(* Logix 5000 project; controller cal1615 1756-L62 rev 20.11; software revision 20.05; part 4 of 81 *)

ADD_ON_INSTRUCTION sys_PIDE   (* revision 1.0, vendor Rockwell Automation *)
VAR_IN_OUT
   Autotune_Tag : PIDE_AUTOTUNE; {required}
END_VAR
VAR_INPUT
   ControlAction : BOOL; {required}
END_VAR
VAR_OUTPUT
   CV : REAL; {access Read Only, required}
END_VAR
VAR_INPUT
   CVMax : REAL; {required}
   CVMin : REAL; {required}
END_VAR
VAR_OUTPUT
   Error : REAL; {access Read Only, required}
END_VAR
VAR_INPUT
   Manual_CV : REAL; {required}
   Manual_Mode : BOOL; {required}
END_VAR
VAR_IN_OUT
   PIDE_Tag : PID_ENHANCED; {required}
END_VAR
VAR_INPUT
   PV : REAL; {required}
   PVMax : REAL; {required}
   PVMin : REAL; {required}
   SP : REAL; {required}
END_VAR
VAR
   BAND_01 : FBD_BOOLEAN_AND := (In1 := 1, In2 := 1, In3 := 1, In4 := 1, In5 := 1, In6 := 1, In7 := 1, In8 := 1);
   BNOT_01 : FBD_BOOLEAN_NOT := (In := 1);
   BOR_01 : FBD_BOOLEAN_OR;
   PIDE_Tag_local : PID_ENHANCED := (PVEUMax := 100.0, SPHLimit := 100.0, RatioProg := 1.0, RatioOper := 1.0, RatioHLimit := 1.0, RatioLLimit := 1.0, CVEUMax := 100.0, CVHLimit := 100.0, PVEDerivative := 1, RTSTime := 1);
   TONR_01 : FBD_TIMER;
   PIDE_Tag_01 : PID_ENHANCED := (PVEUMax := 100.0, SPHLimit := 100.0, RatioProg := 1.0, RatioOper := 1.0, RatioHLimit := 1.0, RatioLLimit := 1.0, CVEUMax := 100.0, CVHLimit := 100.0, PVEDerivative := 1, RTSTime := 1);
   BOR_02 : FBD_BOOLEAN_OR;
   TONR_02 : FBD_TIMER;
   BNOT_02 : FBD_BOOLEAN_NOT := (In := 1);
   BAND_02 : FBD_BOOLEAN_AND := (In1 := 1, In2 := 1, In3 := 1, In4 := 1, In5 := 1, In6 := 1, In7 := 1, In8 := 1);
   __l01DD22F71981FEA5 : REAL;
   __l01DD6E4F1981CCC4 : REAL;
   __l01DD12571981E08E : BOOL;
   __l01DD3F0D1981A0DE : REAL;
   __l01DD266519818F93 : BOOL;
   __l01DD4A391981B409 : REAL;
   __l01DD3B8019819839 : REAL;
   __l01DD359A1981A1AC : REAL;
   __l01DD70B31981916B : REAL;
END_VAR

ROUTINE Logic   (* function block diagram *)
   SHEET 1
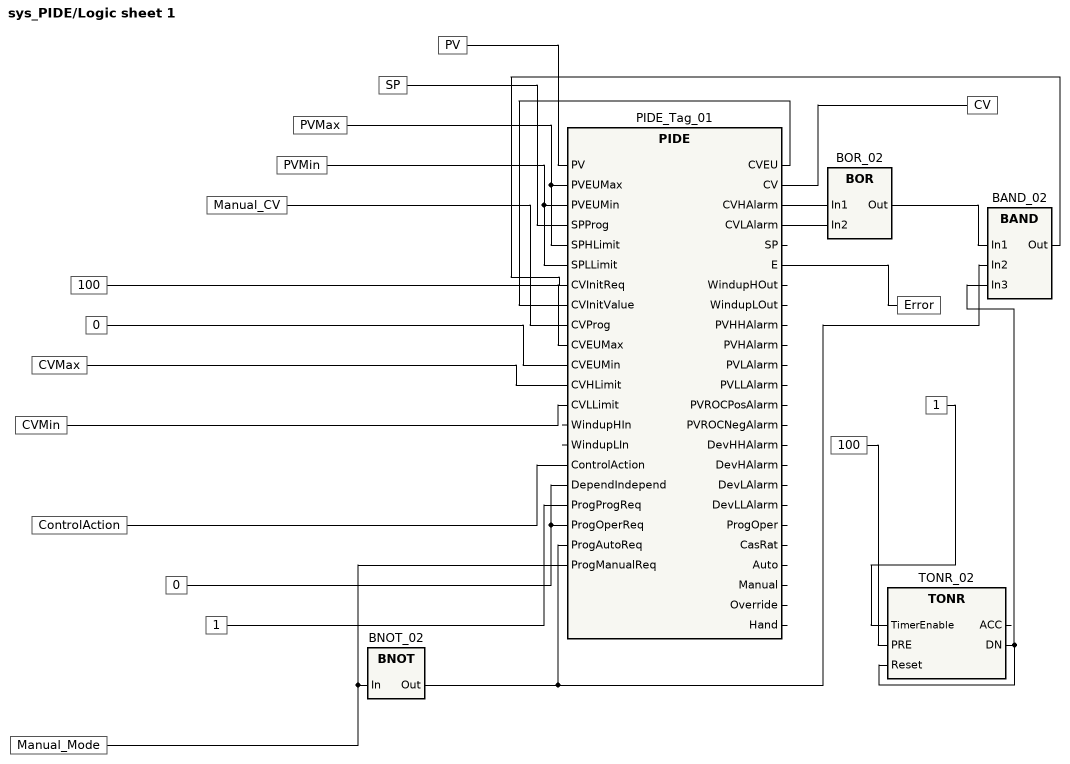
   BNOT_02 : BNOT(In := Manual_Mode);
   PIDE_Tag_01 : PIDE(PV := PV, PVEUMax := PVMax, PVEUMin := PVMin, SPProg := SP, SPHLimit := PVMax, SPLLimit := PVMin, CVInitReq := BAND_02.Out {feedback}, CVInitValue := PIDE_Tag_01.CVEU, CVProg := Manual_CV, CVEUMax := 100, CVEUMin := 0, CVHLimit := CVMax, CVLLimit := CVMin, ControlAction := ControlAction, DependIndepend := 0, ProgProgReq := 1, ProgOperReq := 0, ProgAutoReq := BNOT_02.Out, ProgManualReq := Manual_Mode);   // unwired pins: WindupHIn WindupLIn SP WindupHOut WindupLOut PVHHAlarm PVHAlarm PVLAlarm PVLLAlarm PVROCPosAlarm PVROCNegAlarm DevHHAlarm DevHAlarm DevLAlarm DevLLAlarm ProgOper CasRat Auto Manual Override Hand
   BOR_02 : BOR(In1 := PIDE_Tag_01.CVHAlarm, In2 := PIDE_Tag_01.CVLAlarm);
   Error := PIDE_Tag_01.E;
   CV := PIDE_Tag_01.CV;
   BAND_02 : BAND(In1 := BOR_02.Out, In2 := BNOT_02.Out, In3 := TONR_02.DN {feedback});
   TONR_02 : TONR(TimerEnable := 1, PRE := 100, Reset := TONR_02.DN);   // unwired pins: ACC
END_ROUTINE
END_ADD_ON_INSTRUCTION

ADD_ON_INSTRUCTION sys_Ramp   (* revision 1.0, vendor Rockwell Automation *)
// System Block
// Ramp
VAR_INPUT
   IN_accel_rate : REAL; {required}   // Input Parameter Accel Ramp x/second
   IN_decel_rate : REAL; {required}   // Input Parameter Decel Ramp x/second
   IN_last_scan_s : REAL; {required}   // Input Parameter Last Scan seconds
END_VAR
VAR_IN_OUT
   IN_OUT_ramped_setpoint : REAL; {required}   // Input Output Parameter Ramped Setpoint
END_VAR
VAR_INPUT
   IN_target_setpoint : REAL; {required}   // Input Parameter Targetet Setpoint
END_VAR
VAR
   local_last_scan_ms : DINT;
   p01r03_last_scan_ms : DINT;
END_VAR

ROUTINE Logic   (* ladder *)
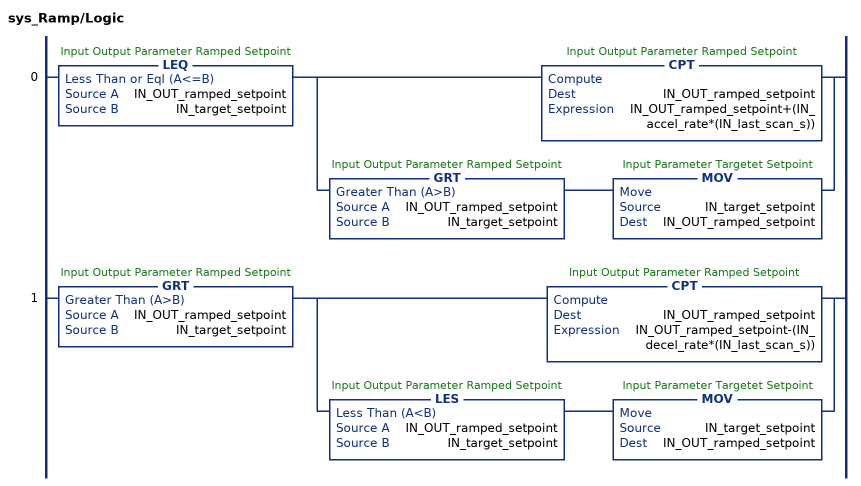
   0: LEQ(IN_OUT_ramped_setpoint,IN_target_setpoint)[CPT(IN_OUT_ramped_setpoint,IN_OUT_ramped_setpoint+(IN_accel_rate*(IN_last_scan_s))) ,GRT(IN_OUT_ramped_setpoint,IN_target_setpoint) MOV(IN_target_setpoint,IN_OUT_ramped_setpoint) ];
   1: GRT(IN_OUT_ramped_setpoint,IN_target_setpoint)[CPT(IN_OUT_ramped_setpoint,IN_OUT_ramped_setpoint-(IN_decel_rate*(IN_last_scan_s))) ,LES(IN_OUT_ramped_setpoint,IN_target_setpoint) MOV(IN_target_setpoint,IN_OUT_ramped_setpoint) ];
END_ROUTINE
END_ADD_ON_INSTRUCTION

ADD_ON_INSTRUCTION SYS_RPM_TO_SPEED   (* revision 1.0 *)
VAR_INPUT
   IN_gear_ratio : REAL; {required}   // Gear Ratio
   IN_roll_diameter : REAL; {required}   // Roll Diameter
   IN_vfd_fb_rpm : REAL; {required}   // VFD Feedback in RPM
END_VAR
VAR_OUTPUT
   OUT_surface_speed_fb : REAL; {access Read Only, required}   // Roll Surface Speed Feedback
END_VAR
VAR
   no_diameter : BOOL;
END_VAR

ROUTINE Logic   (* ladder *)
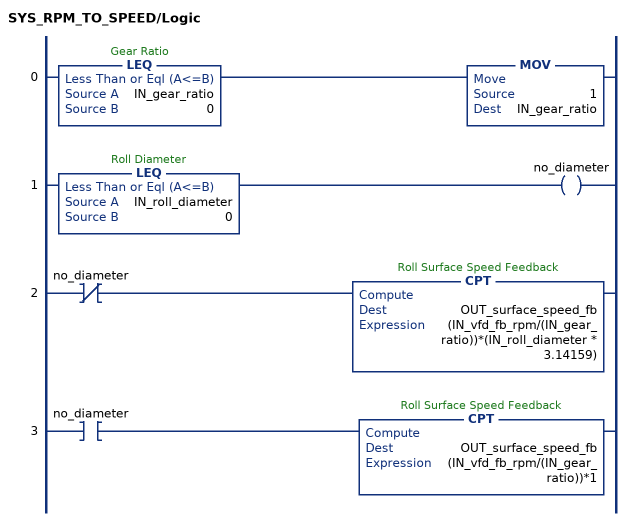
   0: LEQ(IN_gear_ratio,0)MOV(1,IN_gear_ratio);
   1: LEQ(IN_roll_diameter,0)OTE(no_diameter);
   2: XIO(no_diameter)CPT(OUT_surface_speed_fb,(IN_vfd_fb_rpm/(IN_gear_ratio))*(IN_roll_diameter * 3.14159));
   3: XIC(no_diameter)CPT(OUT_surface_speed_fb,(IN_vfd_fb_rpm/(IN_gear_ratio))*1);
END_ROUTINE
END_ADD_ON_INSTRUCTION

ADD_ON_INSTRUCTION SYS_SCP   (* revision 1.0 *)
VAR_INPUT
   Input : REAL; {required}
   Input_Min : REAL; {required}
   Input_Max : REAL; {required}
   Output_Min : REAL; {required}
   Output_Max : REAL; {required}
END_VAR
VAR_OUTPUT
   Output : REAL; {access Read Only, required}
   Fault : BOOL; {access Read Only}
END_VAR
VAR
   m : REAL;
   b : REAL;
   X1 : REAL;
   X2 : REAL;
   Y1 : REAL;
   Y2 : REAL;
   X3 : REAL;
   Y3 : REAL;
END_VAR

ROUTINE Logic   (* ladder *)
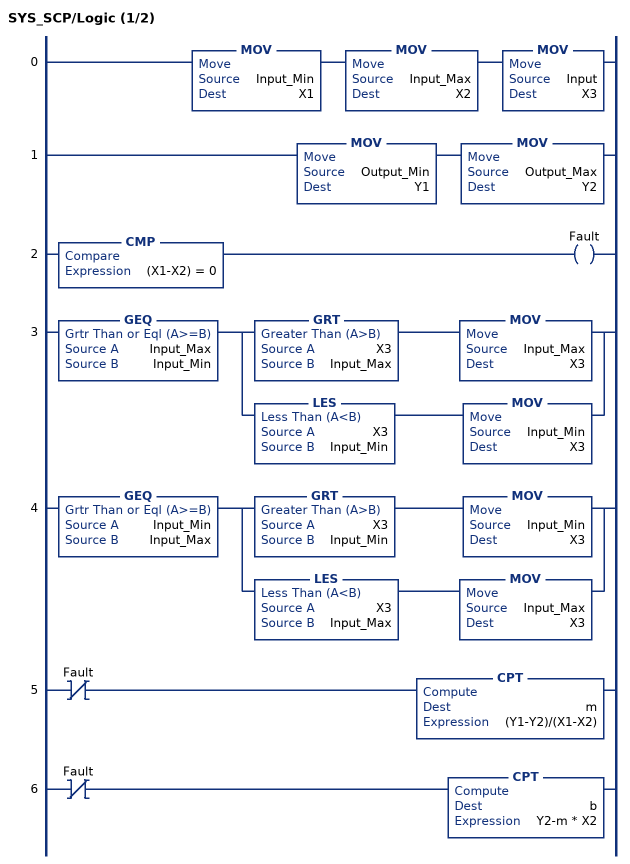
   0: MOV(Input_Min,X1)MOV(Input_Max,X2)MOV(Input,X3);
   1: MOV(Output_Min,Y1)MOV(Output_Max,Y2);
   2: CMP((X1-X2) = 0)OTE(Fault);
   3: GEQ(Input_Max,Input_Min)[GRT(X3,Input_Max) MOV(Input_Max,X3) ,LES(X3,Input_Min) MOV(Input_Min,X3) ];
   4: GEQ(Input_Min,Input_Max)[GRT(X3,Input_Min) MOV(Input_Min,X3) ,LES(X3,Input_Max) MOV(Input_Max,X3) ];
   5: XIO(Fault)CPT(m,(Y1-Y2)/(X1-X2));
   6: XIO(Fault)CPT(b,Y2-m * X2);
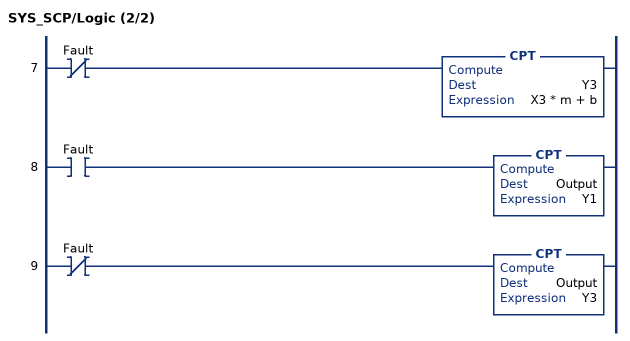
   7: XIO(Fault)CPT(Y3,X3 * m + b);
   8: XIC(Fault)CPT(Output,Y1);
   9: XIO(Fault)CPT(Output,Y3);
END_ROUTINE
END_ADD_ON_INSTRUCTION

ADD_ON_INSTRUCTION SYS_SPEED_TO_VFD   (* revision 1.0 *)
VAR_INPUT
   IN_gear_ratio : REAL; {required}   // Gear Ratio
   IN_roll_diameter : REAL; {required}   // Roll Diameter
   IN_selected_speed : REAL; {required}   // Selected Speed
END_VAR
VAR_OUTPUT
   OUT_surface_speed_rpm : REAL; {access Read Only, required}   // RPM to VFD
END_VAR

ROUTINE Logic   (* ladder *)
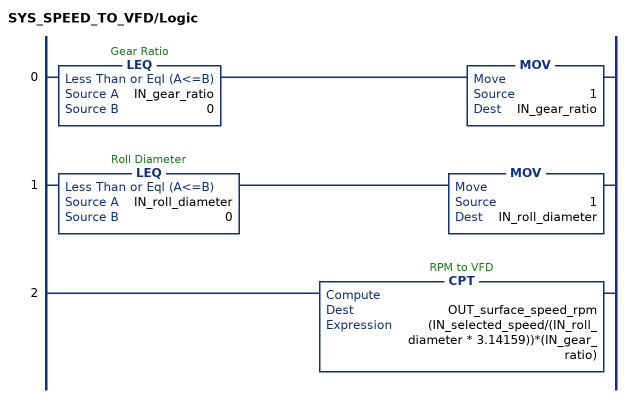
   0: LEQ(IN_gear_ratio,0)MOV(1,IN_gear_ratio);
   1: LEQ(IN_roll_diameter,0)MOV(1,IN_roll_diameter);
   2: CPT(OUT_surface_speed_rpm,(IN_selected_speed/(IN_roll_diameter * 3.14159))*(IN_gear_ratio));
END_ROUTINE
END_ADD_ON_INSTRUCTION

ADD_ON_INSTRUCTION SYS_Toggle   (* revision 1.0 *)
VAR_INPUT
   in_pb : BOOL; {required}   // IN: Momentary On PB
END_VAR
VAR_IN_OUT
   out_state : BOOL; {required}   // OUT: State
END_VAR
VAR_INPUT
   toggle_state : BOOL; {visible}
END_VAR
VAR
   ons : DINT;
        .1   // One Shots
   toggle_select_deselct : BOOL;   // Toggle Select/Deselect
END_VAR

ROUTINE Logic   (* ladder *)
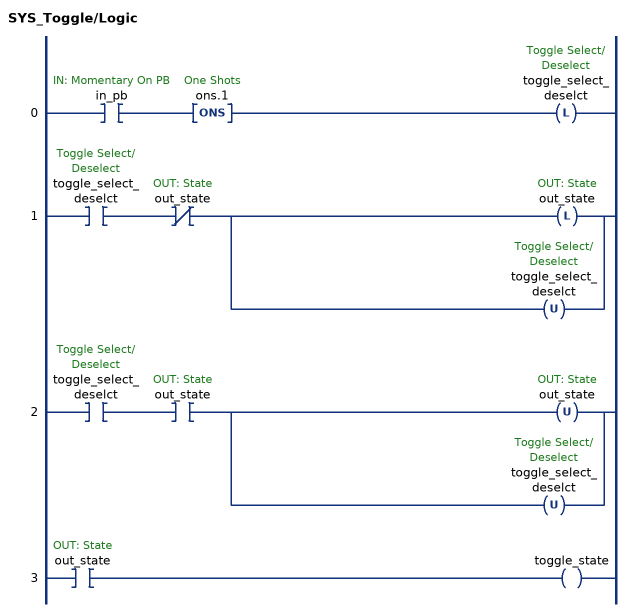
   0: XIC(in_pb)ONS(ons.1)OTL(toggle_select_deselct);
   1: XIC(toggle_select_deselct)XIO(out_state)[OTL(out_state) ,OTU(toggle_select_deselct) ];
   2: XIC(toggle_select_deselct)XIC(out_state)[OTU(out_state) ,OTU(toggle_select_deselct) ];
   3: XIC(out_state)OTE(toggle_state);
END_ROUTINE
END_ADD_ON_INSTRUCTION

VAR_GLOBAL   (* controller tags *)
   aaa_aaa_temp : BOOL;
        .DATA[0]   // Input Zone 2 Recirc VFD Status Word
        .DATA[0].0   // Input Zone 2 Recirc VFD Faulted
        .DATA[0].1   // Input Zone 2 Recirc VFD Warning
        .DATA[0].2   // Input Zone 2 Recirc VFD Running Forward
        .DATA[0].3   // Input Zone 2 Recirc VFD Running Reverse
        .DATA[0].4   // Input Zone 2 Recirc VFD Ready
        .DATA[0].5   // Input Zone 2 Recirc VFD Control from Net
        .DATA[0].6   // Input Zone 2 Recirc VFD Reference from Net
        .DATA[0].7   // Input Zone 2 Recirc VFD At Reference
        .DATA[1]   // Input Zone 2 Recirc VFD Speed
        .DATA[2]   // Input Zone 2 Recirc VFD Amps
        .DATA[3]   // Input Zone 2 Recirc VFD Max Hertz
        .DATA[4]   // Input Zone 2 Recirc VFD Motor Nameplate Hertz
        .DATA[5]   // Input Zone 2 Recirc VFD Motor Nameplate RPM
   aaa_eb_ts2 : BOOL;
   aaa_prs : REAL := 60.0;
   AFI : BOOL;   // Always False Bit
   ai_enc_position : ALIAS FOR T000_ENC_Winder:I.Encoder.Position;
   any_jog_wa_permissive : BOOL;   // Winder A Any Jog Permissive
   any_jog_wb_permissive : BOOL;   // Winder B Any Jog Permissive
   AutoT : PIDE_AUTOTUNE := (ProcessType := 5, PVTuneLimit := 100.0, StepSize := 1.0, ATuneAcquired := 1, UsedProcessType := 7, StepSizeUsed := 1.0, AtuneStatus := 16#0000_0005, ATuneFault := 1, ModeInv := 1);
   di_mode_doff : BOOL;   // Doff Mode
   di_mode_run : BOOL;   // Run Mode
   di_request_move_a_to_doff : BOOL;
   di_request_move_a_to_run : BOOL;
   di_request_move_b_to_doff : BOOL;
   di_request_move_b_to_run : BOOL;
   FAULT : BOOL;   // Fault AFI
   FlashBit_500MSec : BOOL;   // Flash Bit 500 MSec
   HMI : BOOL;   // AFI HMI
   IN_ai_lc01 : ALIAS FOR p00_io_winder:2:I.Ch6Data;
   metering_roll : TIMER;
   metering_roll_alarm : TIMER := (PRE := 4500);
   metering_roll_close : TIMER := (PRE := 5000);
   nip_mode_close : BOOL;   // Nip Mode Close
   p00_FlashBit_1Sec : BOOL;   // System Flash Bit 1 Second
   p00_lin_timer_pre_0ms : DINT;
   p00_lin_timer_pre_1s : DINT;
   p00_lin_timer_pre_disc : DINT;
   p00_lin_timer_pre_mcp : DINT;
   p00_lin_timer_pre_ms : DINT;
   p00_lin_timer_pre_ol : DINT;
   p00_pb_lamp_test : BOOL;
   p00_wac : Accumulator;   // Winder Accumulator
   P00_wac_full : BOOL;
   p00_wac_position_pct : REAL;   // Winder Accumulator Carriage Position Filtered [% of Stroke]
   p01_ai_lc_4 : REAL := 153.39998;
   p01_ai_prs : REAL := -0.6399157;   // System Inputs Oxidizer Differential Pressure
   p01_ai_tc : REAL := 220.4;   // System Inputs Oxidizer Inlet Temperature
   p01_di_edge_ctrl_estop_active : BOOL;   // System Digital Input Edge Control Estop Active
   p01_di_estop_1_tripped : BOOL := 1;   // System Digital Input EStop Relay 1 Tripped
   p01_di_estop_2_tripped : BOOL := 1;   // System Digital Input EStop Relay 2 Tripped
   p01_di_estop_reset : BOOL;   // System Digital Inupt Main Operator Panel E-Stop Reset
   p01_di_impreg_estop_active : BOOL;   // System Digital Input Impreg Estop Active
   p01_di_letoff_estop_active : BOOL;   // System Digital Input Letoff Estop Active
   p01_di_lof_acc_estop_active : BOOL;   // System Digital Input Letoff Accumulator Estop Active
   p01_di_main_hmi_estop : BOOL;   // System Digital Inupt Main Operator Panel E-Stop Active
   p01_di_rope_sw_1_active : BOOL;   // System Digital Input Rope Switch 1 Active
   p01_di_rope_sw_2_active : BOOL;   // System Digital Input Rope Switch 2 Active
   p01_di_rope_sw_3_active : BOOL;   // System Digital Input Rope Switch 3 Active
   p01_di_rope_sw_4_active : BOOL;   // System Digital Input Rope Switch 4 Active
   p01_di_rope_sw_5_active : BOOL;   // System Digital Input Rope Switch 5 Active
   p01_di_rope_sw_6_active : BOOL;   // System Digital Input Rope Switch 6 Active
   p01_di_rope_sw_7_active : BOOL;   // System Digital Input Rope Switch 7 Active
   p01_di_rope_sw_8_active : BOOL;   // System Digital Input Rope Switch 8 Active
   p01_di_splice_estop_active : BOOL;   // System Digital Input Splice Press Estop Active
   p01_di_ts2_estop_active : BOOL;   // System Digital Input Tension Stand 2 Estop Active
   p01_di_winder_estop_active : BOOL;   // System Digital Input Winder Estop Active
   p01_dint_to_hmi : DINT[16] := ([0] := 49794, [1] := 3, [6] := 260, [7] := 3, [8] := 5, [9] := 1, [14] := 15533);   // System Dint to HMI
        [0].8   // System Dint to HMI Oxidizer Spare
        [0].9   // System Dint to HMI Oxidizer Ready
        [0].10   // System Dint to HMI Oxidizer Spare
        [0].11   // System Dint to HMI Oxidizer Spare
        [0].12   // System Dint to HMI Oxidizer Spare
        [0].13   // System Dint to HMI Oxidizer Oven Purge Not Used
        [0].14   // System Dint to HMI Oxidizer Process Block Open
        [0].15   // System Dint to HMI Oxidizer Spare 1/3 Fresh Air
        [1]   // Dint to HMI System Mode
        [2].0   // System Dint to HMI Alarms A00: Emergency Stop
        [2].1   // System Dint to HMI Alarms A01: Main HMI Emergency Stop
        [2].2   // System Dint to HMI Alarms A02: Rope Switch 1 Emergency Stop
        [2].3   // System Dint to HMI Alarms A03: Rope Switch 2 Emergency Stop
        [2].4   // System Dint to HMI Alarms A04: Rope Switch 3 Emergency Stop
        [2].5   // System Dint to HMI Alarms A05: Rope Switch 4 Emergency Stop
        [2].6   // System Dint to HMI Alarms A06: Rope Switch 5 Emergency Stop
        [2].7   // System Dint to HMI Alarms A07: Rope Switch 6 Emergency Stop
        [2].8   // System Dint to HMI Alarms A08: Rope Switch 7 Active
        [2].9   // System Dint to HMI Alarms A09: Rope Switch 8 Active
        [2].10   // System Dint to HMI Alarms A10: Edge Control Emergency Stop
        [2].11   // System Dint to HMI Alarms A11: TS2 Emergency Stop
        [2].12   // System Dint to HMI Alarms A12: Winder Emergency Stop
        [2].13   // System Dint to HMI Alarms A13: Letoff Emergency Stop
        [2].14   // System Dint to HMI Alarms A14: Splice Press Emergency Stop
        [2].15   // System Dint to HMI Alarms A15:Letoff Accumulator Emergency Stop
        [2].16   // System Dint to HMI Alarms A16: Impreg Station Emergency Stop
        [2].17   // System Dint to HMI Alarms A17:
        [2].18   // System Dint to HMI Alarms A18:
        [2].19   // System Dint to HMI Alarms A19:
        [2].20   // System Dint to HMI Alarms A20: Oxidizer Communication Fault
        [2].21   // System Dint to HMI Alarms A21: Oxidizer Oven Purge Damper Closed
        [2].22   // System Dint to HMI Alarms A22: Oxidizer Coupling Damper Open
        [2].23   // System Dint to HMI Alarms A23:
        [2].24   // System Dint to HMI Alarms A24: Impreg Supply Fan Comm Fault
        [2].25   // System Dint to HMI Alarms A25: Zone 1 Recirc VFD Comm Fault
        [2].26   // System Dint to HMI Alarms A26: Zone 1 Exhaust VFD Comm Fault
        [2].27   // System Dint to HMI Alarms A27: Zone 2 Recirc VFD Comm Fault
        [2].28   // System Dint to HMI Alarms A28: Zone 2 Exhaust VFD Comm Fault
        [2].29   // System Dint to HMI Alarms A29: Zone 3 Recirc VFD Comm Fault
        [2].30   // System Dint to HMI Alarms A30: Zone 3 Exhaust VFD Comm Fault
        [2].31   // System Dint to HMI Alarms A31: Letoff A VFD Comm Fault
        [3].0   // System Dint to HMI Alarms A32:Letoff B VFD Comm Fault
        [3].1   // System Dint to HMI Alarms A33:Letoff Turret VFD Comm Fault
        [3].2   // System Dint to HMI Alarms A34: Tension Stand 1 VFD Comm Fault
        [3].3   // System Dint to HMI Alarms A35: Metering Roll VFD Comm Fault
        [3].4   // System Dint to HMI Alarms A36: Metering Servo Operator Side Comm Fault
        [3].5   // System Dint to HMI Alarms A37: Metering Servo Drive Side Comm Fault
        [3].6   // System Dint to HMI Alarms A38: Tension Stand 2 VFD Comm Fault
        [3].7   // System Dint to HMI Alarms A39: Slitter VFD Comm Fault
        [3].8   // System Dint to HMI Alarms A40: Winder Turret VFD Comm Fault
        [3].9   // System Dint to HMI Alarms A41: Winder A VFD Comm Fault
        [3].10   // System Dint to HMI Alarms A42: Winder B VFD Comm Fault
        [3].12   // System Dint to HMI Alarms A43:
        [4].0   // System Warnings W00: PLC Low Battery
        [4].1   // System Warnings W01: System Not in Run Mode
        [4].2   // System Warnings W02: Zone 2 Access Door Open
        [4].3   // System Warnings W03:
        [4].4   // System Warnings W04:
        [4].5   // System Warnings W05:Letoff A drive fault
        [4].6   // System Warnings W06:Letoff B drive fault
        [4].7   // System Warnings W07:Letoff turret drive fault
        [4].8   // System Warnings W08:Tension stand 1 drive fault
        [4].9   // System Warnings W09:metering roll drive fault
        [4].10   // System Warnings W10:tension stand 2 drive fault
        [4].11   // System Warnings W11:Slitter driver fault
        [4].12   // System Warnings W12:Winder A drive fault
        [4].13   // System Warnings W13:Winder B drive fault
        [4].14   // System Warnings W14:An active letoff has not been selected
        [4].15   // System Warnings W15:An active winder has not been selected
        [4].16   // System Warnings W16:Letoff turret is not in position
        [4].17   // System Warnings W17:
        [4].18   // System Warnings W18:
        [4].19   // System Warnings W19:
        [4].20   // System Warnings W20:
        [4].21   // System Warnings W21:
        [4].22   // System Warnings W22:
        [4].23   // System Warnings W23:
        [4].24   // System Warnings W24:
        [4].25   // System Warnings W25:
        [4].26   // System Warnings W26:
        [4].27   // System Warnings W27:
        [4].28   // System Warnings W28:
        [4].29   // System Warnings W29:
        [4].30   // System Warnings W30
        [4].31   // System Warnings W31:
        [6].0   // System Dint to HMI PI: Unacknowledged Alarm/Warning Exists
        [6].1   // System Dint to HMI PI: Logout
        [6].2   // System Dint fo HMI Preventive Maintenance Trigger
        [6].3   // System Dint to HMI PI: Line Running
        [6].6   // System Dint to HMI PI: All Fans Stopped
        [6].7   // System Dint to HMI PI: All Fans Stopped
        [6].8   // System Dint to HMI PI: Oven Auto Sequence On
        [7]   // System Dint To HMI Line Mode
        [8]   // System Dint to HMI Oxidizer Status
        [9]   // System Dint to HMI Line Start Sequence Step
        [15]   // System Dint to HMI Thread "Master"
   p01_int_from_oxidizer : INT[10] := ([0] := -15856, [1] := 1, [2] := 210, [3] := 39, [4] := 1581, [5] := 1549, [6] := 249, [7] := 58, [8] := 1552, [9] := 1463); {produced}   // System Oxidizer Int from Oxidizer
        [0].0   // System Oxidizer Iface Int from Oxidizer Combustion Purge Mode
        [0].1   // System Oxidizer Iface Int from Oxidizer Purge Mode
        [0].2   // System Oxidizer Iface Int from Oxidizer Heat Mode
        [0].3   // System Oxidizer Iface Int from Oxidizer Soak Mode
        [0].4   // System Oxidizer Iface Int from Oxidizer Run Mode
        [0].5   // System Oxidizer Iface Int from Oxidizer Bake Mode
        [0].6   // System Oxidizer Iface Int from Oxidizer Fault Mode
        [0].7   // System Oxidizer Iface Int from Oxidizer Shutdown
        [0].8   // System Oxidizer Iface Int from Oxidizer (Spare)
        [0].9   // System Oxidizer Iface Int from Oxidizer Oxidizer Ready
        [0].13   // System Oxidizer Iface Int from Oxidizer Oven Purge
        [0].14   // System Oxidizer Iface Int from Oxidizer Process Block Open
        [0].15   // System Oxidizer Iface Int from Oxidizer 1/3 Flow Fresh Air
        [1].0   // System Oxidizer Iface Int from Oxidizer Oven Purge Damper Closed
        [1].1   // System Oxidizer Iface Int from Oxidizer Heart Beat
        [2]   // System Oxidizer Iface Int from Oxidizer TE-101 Inlet T/C
        [3]   // System Oxidizer Iface Int from Oxidizer Oxidizer Delta Temperature
        [4]   // System Oxidizer Iface Int from Oxidizer TE-103 Chamber T/C
        [5]   // System Oxidizer Iface Int from Oxidizer TE-104 Chamber T/C
        [6]   // System Oxidizer Iface Int from Oxidizer TE-105 Exhaust T/C
        [7]   // System Oxidizer Iface Int from Oxidizer TE-107 Combustion Air T/C
        [8]   // System Oxidizer Iface Int from Oxidizer TE-108 Bed T/C
        [9]   // System Oxidizer Iface Int from Oxidizer TE-109 Bed T/C
   p01_int_to_oxidizer : INT := 1;   // System Oxidizer Int to Oxidizer
        .0   // System Oxidizer Iface Int to Oxidizer Purge Complete
        [0].0   // System Oxidizer Iface Int to Oxidizer Combustion Purge Complete
   p01_param_fan_zero_speed : REAL := 0.1;
   p01_param_heater_hl : REAL := 785.0;   // Machine Parameter Heater HighTemperature Max Limit
   p01_param_master_accel : REAL := 0.5;   // Machine Parameter Master Accel Rate
   p01_param_master_decel : REAL := 2.5;   // Machine Parameter Master Decel Rate
   p01_param_master_jog_accel : REAL := 10.0;   // Machine Parameter Master Jog Acceleration mmpm/s
   p01_param_master_jog_decel : REAL := 20.0;   // Machine Parameter Master Jog Deceleration mmpm/s
   p01_param_master_jog_speed : REAL := 8.0;   // Machine Parameter Master Jog Speed
   p01_param_min_start_tension : REAL := 10.0;
   p01_param_mtr_over_speed_pct : REAL := 7.1999974;   // System Parameter Metering Roll Overspeed [pct]
   p01_param_open_oven_exh_sp : REAL := 300.0;
   p01_param_open_oven_recirc_sp : REAL := 300.0;
   p01_param_open_oven_temp : REAL := 80.0;
   p01_param_oven_timer_presets : DINT[32] := ([1] := 500, [2] := 10000, [3] := 20000, [6] := 5000, [8] := 1000, [9] := 1000, [10] := 1000, [11] := 5000, [14] := 10000, [16] := 1000, [17] := 90000, [18] := 1500, [19] := 1000, [21] := 1000, [22] := 1000, [23] := 2000, [24] := 5000, [25] := 5000, [26] := 15000, [27] := 500, [28] := 30000, [31] := 500);   // System Parameter Oven Timer Presets
        [0]   // System Timer Presets Parameter Oven Motor Starter Fault
        [1]   // System Timer Presets Parameter Oven Motor Starter Temperature Not OK
        [2]   // System Timer Presets Parameter Oven Motor Off while Chamber Temperature is Too High
        [3]   // System Timer Presets Parameter Oven Fan Pressure Low
        [4]   // System Timer Presets Parameter
        [5]   // System Timer Presets Parameter Spare
        [6]   // System Timer Presets Parameter Oven Software High Limit
        [7]   // System Timer Presets Parameter Oven Hardware High Limit - all Burner Safeties
        [8]   // System Timer Presets Parameter TC Failures
        [9]   // System Timer Presets Parameter Man Door Faults
        [10]   // System Timer Presets Parameter LFL Fault-Warning
        [11]   // System Timer Presets Parameter Spare
        [12]   // System Timer Presets Parameter Spare
        [13]   // System Timer Presets Parameter Spare
        [14]   // System Timer Presets Parameter Oven Temperature Deviation Warning
        [15]   // System Timer Presets Parameter Spare
        [16]   // System Timer Presets Parameter Filter Dirty Warning
        [17]   // System Timer Presets Parameter Zone in Manual Warning
        [18]   // System Timer Presets Parameter Zone High Pressure
        [19]   // System Timer Presets Parameter Filter Dirty Delay
        [20]   // System Timer Presets Parameter Spare
        [21]   // System Timer Presets Parameter State 3 Dwell
        [22]   // System Timer Presets Parameter Stat 4 Dwell
        [23]   // System Timer Presets Parameter State 7 Dwell
        [24]   // System Timer Presets Parameter State 8 Dwell
        [25]   // System Timer Presets Parameter Spare
        [26]   // System Timer Presets Parameter Oven Auto Fan Start Sequence Stall
        [27]   // System Timer Presets Parameter Spare
        [28]   // System Timer Presets Parameter Oven Shutdown Temperature Delay
        [29]   // System Timer Presets Parameter Spare
        [30]   // System Timer Presets Parameter Spare
        [31]   // System Timer Presets Parameter Spare
   p01_param_process_air_hl : REAL := 500.0;   // Machine Parameter Process Air High Limit
   p01_param_process_air_max : REAL := 480.0;   // Machine Parameter Process Air High Temperature Max Setpoint Limit
   p01_param_slow_speed_sp : REAL := 2.0;   // System Parameters Slow Speed Setpoint
   p01_param_start_delay : REAL := 6.0;   // Machine Parameter Start Delay
   p01_param_temp_limit : REAL := 120.0;   // Machine Parameter Maximum Temperature for Fan Operation
   p01_param_tension_deviation : REAL := 5.0;
   p01_param_turret_dia_ft : REAL := 3.2;
   p01_r15_footage_ft : REAL;   // System Customer Footage Counter
   p01_real_to_hmi : REAL[112] := ([1] := 8.0, [11] := 210.0, [12] := 40.0, [13] := 1583.0, [14] := 1549.0, [15] := 250.0, [16] := 58.0, [17] := 1557.0, [18] := 1459.0, [19] := 4157.8765);   // System Real to HMI
        [0]   // System Real to HMI Master Ramped Speed
        [1]   // System Real to HMI Master Jog Speed
        [2]   // System Real to HMI Footage
   p01_recipe_active : recipe := (name := '20210820_rcp.csv', master_line_speed := 10.0, zone_1.recirc_sp := 1100.0, zone_1.exhaust_sp := 900.0, zone_1.temp_sp := 260.0, zone_2.recirc_sp := 1100.0, zone_2.exhaust_sp := 900.0, zone_2.temp_sp := 260.0, zone_3.recirc_sp := 1300.0, zone_3.exhaust_sp := 900.0, zone_3.temp_sp := 60.0, line_speed_sp := 8.0, letoff_tension_sp := 15.0, acc_tension_sp := 50.0, acc_fill_pressure_sp := 10.0, acc_counter_pressure_sp := 10.0, cure_time_sp := 55.0, platen_temp_sp := 450.0, impreg_gap_sp := 0.016, impreg_supply_speed_sp := 1200.0, ts1_tension_sp := 50.0, slitter_speed_sp := 6.0, adv_cooling_temp_sp := 60.0, ts2_tension_sp := 60.0, lower_poly_tension_sp := 2.0, lower_poly_b_tension_sp := 2.0, upper_poly_tension_sp := 2.0, upper_poly_b_tension_sp := 2.0, winder_tension_sp := 70.0, winder_torque_sp := 100.0, tension_deviation_sp := 6.0);   // Active Recipe
   p01_sys_enc : SYS_ENC := (IN_State := 33, OUT_Status := 5);   // System Encoder
   p01_sys_lc : Limit_Clamp := (max := 100.0);   // Zone 1 Misc Control Limit Clamp
   p01_sys_scp : SYS_SCP := (Input := 12904.0, Input_Max := 30840.0, Output_Max := 50.0, Output := 20.920883);   // System Scaling
   p01r01 : routine := (comment := 7);
   p01r02 : routine := (comment := -1073741569);   // System Misc Control
        .FAULT.0   // System Misc Control Impreg Supply Fan VFD Comm Faulted
        .FAULT.1   // System Misc Control Zone 1 Recirc VFD Comm Faulted
        .FAULT.2   // System Misc Control Zone 1 Exhaust VFD Comm Faulted
        .FAULT.3   // System Misc Control Zone 2 Recirc VFD Comm Faulted
        .FAULT.4   // System Misc Control Zone 2 Exhaust VFD Comm Faulted
        .FAULT.5   // System Misc Control Zone 3 Recirc VFD Comm Faulted
        .FAULT.6   // System Misc Control Zone 3 Exhaust VFD Comm Faulted
        .FAULT.7   // System Misc Control Letoff A VFD Comm Faulted
        .FAULT.8   // System Misc Control Letoff B VFD Comm Faulted
        .FAULT.9   // System Misc Control Letoff Turret VFD Comm Faulted
        .FAULT.10   // System Misc Control Tension Stand 1 VFD Comm Faulted
        .FAULT.11   // System Misc Control Metering Roll VFD Comm Faulted
        .FAULT.12   // System Misc Control Metering Servo Operator Side Comm Faulted
        .FAULT.13   // System Misc Control Metering Roll Drive Side Comm Faulted
        .FAULT.14   // System Misc Control Tension Stand 2 VFD Comm Faulted
        .FAULT.15   // System Misc Control Slitter VFD Comm Faulted
        .FAULT.16   // System Misc Control Winder Turret VFD Comm Faulted
        .FAULT.17   // System Misc Control Winder A VFD Comm Faulted
        .FAULT.18   // System Misc Control Winder B VFD Comm Faulted
        .WARNING.0   // System Misc Control PLC Low Battery
        .UNACK_FAULT   // System Misc Control Unaknowledged Fault Exists
        .UNACK_WARNING   // System Misc Control Unaknowledged Warning Exists
   p01r02_all_fans_stopped : BOOL;   // System Misc Control All Fans Stopped
   p01r02_batch_run_time : DINT := 1;   // System Misc Control Batch Minutes
   p01r02_batch_run_time_hrs : DINT := 15533;   // System Misc Control Batch Hours
   p01r02_do_buzzer : BOOL;   // System Outputs Buzzer
   p01r02_do_buzzer_LINE : BOOL;
   p01r02_do_green_stack_light_lel : BOOL := 1;   // System Outputs Green Stack Light
   p01r02_do_green_stack_light_LINE : BOOL;
   p01r02_do_horn : BOOL;   // System Outputs Horn
   p01r02_do_red_stack_light : BOOL;   // System Outputs Red Stack Light
   p01r02_do_red_stack_light_LINE : BOOL;
   p01r02_do_yellow_stack_light : BOOL;   // System Outputs Yellow Stack Light
   p01r02_do_yellow_stack_light_LINE : BOOL;
   p01r02_ethernet_comm : DINT := 524287;
        .0   // System Misc Control Impreg Supply Fan VFD Communication Ok
        .1   // System Misc Control Zone 1 Recirc VFD Communication Ok
        .2   // System Misc Control Zone 1 Exhaust VFD Communication Ok
        .3   // System Misc Control Zone 2 Recirc VFD Communication Ok
        .4   // System Misc Control Zone Exhaust VFD Communication Ok
        .5   // System Misc Control Zone 3 Recirc VFD Communication Ok
        .6   // System Misc Control Zone 3 Exhaust VFD Communication Ok
        .7   // System Misc Control Letoff A VFD Communication Ok
        .8   // System Misc Control Letoff B VFD Communication Ok
        .9   // System Misc Control Letoff Turret VFD Communication Ok
        .10   // System Misc Control Tension Stand 1 VFD Communication Ok
        .11   // System Misc Control Metering Roll VFD Communication Ok
        .12   // System Misc Control Metering Servo Operator Side Communication Ok
        .13   // System Misc Control Metering Servo Drive Side Communication Ok
        .14   // System Misc Control Tension Stand 2 VFD Communication Ok
        .15   // System Misc Control Slitter VFD Communication Ok
        .16   // System Misc Control Winder Turret VFD Communication Ok
        .17   // System Misc Control Winder A VFD Communication Ok
        .18   // System Misc Control Winder B VFD Communication Ok
   p01r02_fault_exists : BOOL;
   p01r02_flash_bit : BOOL;   // System Misc Control Flash Bit
   p01r02_flash_timer_off : TIMER := (PRE := 1000);   // System Misc Control Flash Timer Off
   p01r02_flash_timer_on : TIMER := (PRE := 1000);   // System Misc Control Flash Timer On
   p01r02_horn : BOOL;
   p01r02_plc_faults : DINT := 16;   // System Misc Control PLC Faults
        .10   // System Misc Control PLC Fault 10 Low Battery Warning
   p01r02_plc_scan_time : DINT := 30556;   // System PLC Scan Time
   p01r02_plc_scan_time_in_sec : REAL := 0.030376;   // System PLC Scan Time in Seconds
   p01r02_timer_batch : TIMER := (PRE := 60000);   // System Misc Control Batch Timer Seconds
   p01r02_timer_fault : TIMER[25];   // System Misc Control Fault Dwell Timer
   p01r02_timer_half_second_off : TIMER := (PRE := 300, ACC := 303, EN := 1, DN := 1);   // System Misc Control Timer Second Pulse Off
   p01r02_timer_half_second_on : TIMER := (PRE := 300);   // System Misc Control Timer 1/2 Second Pulse On
   p01r02_timer_second : TIMER[2] := ([0].PRE := 1000, [0].ACC := 881, [0].EN := 1, [0].TT := 1, [1].PRE := 1000);   // System Misc Control Timer Second Pulse
   p01r02_timer_warning : TIMER[4];   // System Misc Control Warning Delay
   p01r02_unack_fault : BOOL;   // System Misc Control Unacknowledged Fault Exists
   p01r02_unack_warning : BOOL;   // System Misc Control Unacknowledged Warning Exists
   p01r02_vfd_comm_2 : DINT[50] := ([0] := 16897, [1] := 16897, [2] := 16897, [3] := 16897, [4] := 16897, [5] := 16897, [6] := 16897, [7] := 16897, [8] := 16897, [9] := 16897, [10] := 16897, [11] := 16897, [12] := 16897, [13] := 16897, [14] := 16897, [15] := 16897, [16] := 16897, [17] := 16897, [18] := 16897);
        [11]   // System Misc Control Comm Status
   p01r02_warnings_exists : BOOL;
   p01r03 : routine := (comment := -1073741793);   // System Inputs
        .UNACK_FAULT   // System Input Unaknowledged Fault Exists
        .UNACK_WARNING   // System Inputs Unaknowledged Warning Exists
   p01r03_lc3_ave_ctrl : CONTROL := (LEN := 19, POS := 18, EN := 1, DN := 1);
   p01r03_oxidizer_prs : SYS_SCP := (Input := 11631.0, Input_Max := 30840.0, Output_Min := -2.5, Output_Max := 2.5, Output := -0.61429965);   // System Inputs Oxidizer Differential Pressure Scaling
   p01r03_prs_input_max : REAL := 30840.0;
   p01r03_prs_input_min : REAL;
   p01r03_prs_output_max : REAL := 2.5;
   p01r03_prs_output_min : REAL := -2.5;
   p01r03_timer_fault : TIMER[4];   // System Input Fault Delay
   p01r03_timer_warning : TIMER[4];   // System Input Warning Delay
        [0]   // System Analog Input Warning Delay
   p01r04 : routine := (comment := -1073741793);   // System Outputs
        .UNACK_FAULT   // System Output Unaknowledged Fault Exists
        .UNACK_WARNING   // System Ouputs Unaknowledged Warning Exists
   p01r04_LFL_warning : BOOL;   // System Misc Control LFL Warning
   p01r04_Temp_deviation_warning : BOOL := 1;   // System Misc Control Temperature Deviation Warning
   p01r04_timer_fault : TIMER[4];   // System Output Fault Delay
   p01r04_timer_warning : TIMER[4];   // System Output Warning Delay
   p01r05 : routine := (comment := -1073741761);   // System Dint to HMI
        .UNACK_FAULT   // System Dint to HMI Unaknowledged Fault Exists
        .UNACK_WARNING   // System Dint to HMI Unaknowledged Warning Exists
   p01r05_enc : SYS_ENC;   // System Dint to HMI Encoder
   p01r05_timer_fault : TIMER[4];   // System Dint to HMI Fault Delay
   p01r05_timer_warning : TIMER[4];   // System Dint to HMI Warning Delay
        [0]   // System Dint to HMI Warning Delay
   p01r06 : routine := (comment := -1073741572);   // System Real to HMI
        .UNACK_FAULT   // System Real to HMI Unaknowledged Fault Exists
        .UNACK_WARNING   // System Real to HMI Unaknowledged Warning Exists
   p01r06_timer_fault : TIMER[4];   // System Real to HMI Fault Delay
   p01r06_timer_warning : TIMER[4];   // System Real to HMI Warning Delay
   p01r07 : routine := (comment := -1073741761);   // System Alarms
        .UNACK_FAULT   // System Alarms Unaknowledged Fault Exists
        .UNACK_WARNING   // System Alarms Unaknowledged Warning Exists
   p01r07_timer_fault : TIMER[4];   // System Alarms Fault Delay
   p01r07_timer_warning : TIMER[4];   // System Alarms Warning Delay
   p01r08 : routine := (comment := -1073741761);   // System Warnings
        .UNACK_FAULT   // System Warnings Unaknowledged Fault Exists
        .UNACK_WARNING   // System Warnings Unaknowledged Warning Exists
   p01r08_timer_fault : TIMER[4];   // System Warnings Fault Delay
   p01r08_timer_warning : TIMER[4];   // System Warnings Warning Delay
   p01r09 : routine := (comment := -1073741009, oneshot := 24);   // System Modes
        .FAULT.0   // System Modes Emergency Stop
        .FAULT.1   // System Modes Main HMI Emergency Stop
        .FAULT.2   // System Modes Rope Switch 1 Emergency Stop
        .FAULT.3   // System Modes Rope Switch 2 Emergency Stop
        .FAULT.4   // System Modes Rope Switch 3 Emergency Stop
        .FAULT.5   // System Modes Rope Switch 4 Emergency Stop
        .FAULT.6   // System Modes Rope Switch 5 Emergency Stop
        .FAULT.7   // System Modes Rope Switch 6 Emergency Stop
        .FAULT.8   // System Modes Rope Switch 7 Active
        .FAULT.9   // System Modes Rope Switch 8 Active
        .FAULT.10   // System Modes Edge Control Emergency Stop
        .FAULT.11   // System Modes Tension Stand 2 Emergency Stop
        .FAULT.12   // System Modes Winder Emergency Stop
        .FAULT.13   // System Modes Letoff Emergency Stop
        .FAULT.14   // System Modes Splice Press Emergency Stop
        .FAULT.15   // System Modes Letoff Accumulator Emergency Stop
        .FAULT.16   // System Modes Impreg Emergency Stop
        .FAULT.17   // System Modes Upper Poly Letoff OP Station B: Emergency Stop
        .FAULT.18   // System Modes Lower Poly Letoff OP Station B: Emergency Stop
        .WARNING.0   // System Modes System Not in Run Mode
        .WARNING.1   // System Modes Zone 2 Access Door Open
        .UNACK_FAULT   // System Modes Unaknowledged Fault Exists
        .UNACK_WARNING   // System Modes Unaknowledged Warning Exists
   p01r09_estop_ok : BOOL := 1;   // System Modes Estop Dwell OK
   p01r09_mode_jog : BOOL;   // System Modes Jog Mode
   p01r09_mode_run : BOOL := 1;   // System Modes All Modes Run Mode
   p01r09_mode_thread : BOOL := 1;   // System Modes Thread Mode
   p01r09_open_oven : BOOL;
   p01r09_open_oven_toggle : SYS_Toggle;
   p01r09_pb_global_reset : BOOL;   // System Modes PB: Global Fault Reset
   p01r09_pb_line_jog : BOOL;   // System Modes PB: Line Jog Forward
   p01r09_permissive_change : BOOL := 1;   // System Modes Permissive Mode Change
   p01r09_request_line_jog : BOOL;   // System Modes Request Line Jog Forward
   p01r09_stretch_mode : BOOL;
   p01r09_timer_estop_reset : TIMER := (PRE := 1000, ACC := 1026, EN := 1, DN := 1);   // System Modes Estop Reset Dwell
   p01r09_timer_fault : TIMER[20];   // System Modes Fault Delay
   p01r09_timer_global_reset : TIMER := (PRE := 1000);   // System Modes Global Reset Timer
   p01r09_timer_warning : TIMER[4];   // System Modes Warning Delay
   p01r10 : routine := (comment := -1073741569);   // System Annunciators
        .UNACK_FAULT   // System Annunciators Unaknowledged Fault Exists
        .UNACK_WARNING   // System Annunciators Unaknowledged Warning Exists
   p01r10_fault_exists : BOOL;
   p01r10_timer_fault : TIMER[4];   // System Fault Delay
   p01r10_timer_warning : TIMER[4];   // System Warning Delay
   p01r10_unack_fault : DINT;
   p01r10_unack_fault_ex : BOOL;
   p01r10_unack_warn_ex : BOOL;   // System Annunciators Unacknowledged Warning Exists
   p01r10_unack_warning : DINT;   // System Annunciators Unacknowledged Warning Exists
   p01r10_warning_exists : BOOL := 1;
   p01r11 : routine := (comment := -1073741761);   // System Timer Presets
        .UNACK_FAULT   // System Timer Presets Unaknowledged Fault Exists
        .UNACK_WARNING   // System Timer Presets Unaknowledged Warning Exists
   p01r11_timer_fault : TIMER[4];   // System Fault Delay
   p01r11_timer_warning : TIMER[4];   // System Warning Delay
   p01r12 : routine := (comment := -1073741761);   // System Line Accel Decel Control
        .UNACK_FAULT   // System Line Accel Decel Control Unaknowledged Fault Exists
        .UNACK_WARNING   // System Line Accel Decel Control Unaknowledged Warning Exists
   p01r12_accel_rate : REAL := 0.5;   // Machine Parameter Master Jog Acceleration mmpm/s
   p01r12_decel_rate : REAL := 2.5;   // Machine Parameter Master Jog Deceleration mmpm/s
   p01r12_line_at_speed : BOOL;
   p01r12_master_acel_decel_ramp : SYS_ACC_DEC_RAMP := (IN_param_master_accel_rate := 0.5, IN_param_master_decel_rate := 2.5, IN_last_scan_s := 0.030358);   // System Line Accel Decel Control Ramp
   p01r12_master_ramped_speed : REAL;   // System Line Accel Decel Control Master Ramped Speed
   p01r12_ramped_setpoint : REAL;   // System Line Accel Decel Control Ramped Setpoint
   p01r12_request_any_jog_thread : BOOL;   // System Line Accel Decel Control Request Any Jog/Thread
   p01r12_selected_line_speed : REAL;   // System Line Accel Decel Control Selected Line Speed
   p01r12_timer_fault : TIMER[8];   // System Line Start Sequence Fault Delay
   p01r12_timer_warning : TIMER[8];   // System Line Start Sequence Warning Delay
   p01r12_zero_line_speed : BOOL := 1;   // System Line Accel Decel Control Line Speed at Zero
   p01r13 : routine := (comment := -1073708945);   // System Line Start Sequence
        .FAULT.0   // System Line Start Sequence
        .FAULT.1   // System Line Start Sequence
        .UNACK_FAULT   // System Line Start Sequence Unaknowledged Fault Exists
        .UNACK_WARNING   // System Line Start Sequence Unaknowledged Warning Exists
   p01r13_check_status : BOOL;   // System Line Start Sequence Check Status
   p01r13_check_status_time : REAL := 5750.0;   // System Line Start Sequence Check Status
   p01r13_check_status_timer : TIMER := (PRE := 15000);   // System Line Start Sequence Check Status Timer
   p01r13_check_tension : TIMER;   // System Line Start Sequence Check Tension
   p01r13_letoff_tension_ok : BOOL;   // System Line Start Sequence Letoff Tension Ok
   p01r13_LFL_stop : BOOL;   // System Line Stop from LFL
   p01r13_line_running : BOOL;   // System Line Start Sequence Line Running
   p01r13_line_slow_ramp : BOOL;   // System Line Start Sequence Start Line to Slow Speed
   p01r13_line_start : SYS_ENC := (IN_State := 3, OUT_Status := 1);   // System Line Start Sequence Encoder
   p01r13_oven_temp_ok : BOOL := 1;   // System Line Start Sequence Oven Temperature Ready
   p01r13_pb_start : BOOL;   // System Line Start Sequence PB: Line Start
   p01r13_pb_stop : BOOL;   // System Line Start Sequence PB: Line Stop
   p01r13_permissive_drives : BOOL := 1;   // System Line Start Sequence Permissive Drives
   p01r13_permissive_line_run : BOOL := 1;   // System Line Start Sequence Permissive Line Run
   p01r13_permissive_oven : BOOL := 1;   // System Line start Sequence Permissive Ovens
   p01r13_permissive_oxidizer : BOOL := 1;   // System Line Start Sequence Permissive Oxidizer
   p01r13_request_run : BOOL;   // System Line Start Sequence Request Run
   p01r13_request_stop : BOOL;   // System Line Start Sequence Request Stop
   p01r13_state : DINT := 3;   // System Line Start Sequence Sequencer Step
        .0   // System Line Start Sequence State 0 One Step per Scan
        .1   // System Line Start Sequence State 1 Idle
        .2   // System Line Start Sequence State 2 Initiate Start
        .3   // System Line Start Sequence State 3 Pre-Run Warning
        .4   // System Line Start Sequence State 4 Start and Ramp to Slow Speed
        .5   // System Line Start Sequence State 5 Accelerate to Setpoint in Stretch
        .6   // System Line Start Sequence State 6 Auto Switchover to Tension Control
        .7   // System Line Start Sequence State 7 Run
        .8   // System Line Start Sequence State 8 Initiate Normal Stop
        .9   // System Line Start Sequence State 9 Cycle Complete
   p01r13_status : DINT := 1;   // System Line Start Sequence Encoded Step
   p01r13_system_mode_run : BOOL := 1;   // System Line Start Sequence All Drive Sections in Run Mode
   p01r13_temperature_status_check : TIMER := (PRE := 10000, ACC := 10020, EN := 1, DN := 1);   // System Line Start Sequence Temperature Check
   p01r13_tension_ok : BOOL;   // System Line Start Sequence Slow Speed Tension Ok
   p01r13_timer_fault : TIMER[8];   // System Line Start Sequence Fault Dwell Timer
   p01r13_timer_line_start_warning_dwell : TIMER := (PRE := 6000);   // System Line Start Sequence Pre Start Warning Dwell Timer
   p01r13_timer_line_stop_dwell : TIMER := (PRE := 60000);   // System Line Start Sequence Line Stop Dwell Timer
   p01r13_timer_switch_to_stretch_dwell : TIMER;   // System Line Start Sequence Setpoint Stretch to Tension Dwell Timer
   p01r13_timer_warning : TIMER[8];   // System Line Start Sequence Warning Dwell Timer
   p01r13_ts1_tension_ok : BOOL;   // System Line Start Sequence TS 1 Tension Ok
   p01r13_ts2_tension_ok : BOOL;   // System Line Start Sequence TS 2 Tension Ok
   p01r13_winder_tension_ok : BOOL;   // System Line Start Sequence Winder Tension Ok
   p01r14 : routine := (comment := -1073741697);
        .FAULT   // System Oxidizer Faults
        .FAULT.0   // System Oxidizer Communication Fault
        .FAULT.1   // System Oxidizer Oven Purge Damper Closed Fault
        .FAULT.2   // System Oxidizer Coupling Damper Open Fault
        .FAULT_ACK   // System Oxidizer Ackn. Faults
        .UNACK_FAULT   // System Oxidizer Unaknowledged Fault Exists
   p01r14_msg_read : MESSAGE;   // System Oxidizer Message Read
        MessageParameters(ServiceCode := 16#0fa2, LocalElement := p01_int_from_oxidizer[0], ...)
   p01r14_msg_read_retry_timer : TIMER := (PRE := 1000);
   p01r14_msg_read_timer : TIMER := (PRE := 200);   // System Oxidizer Read Dwell
   p01r14_msg_write : MESSAGE;   // System Oxidizer Message Write
        MessageParameters(ServiceCode := 16#0faa, LocalElement := p01_int_to_oxidizer, ...)
   p01r14_msg_write_retry_timer : TIMER := (PRE := 1000);   // System Oxidizer Message Retry Timer
   p01r14_msg_write_timer : TIMER := (PRE := 100, ACC := 61, EN := 1, TT := 1);   // System Oxidizer Message Read Dwell
   p01r14_oxidizer_heart_beat_off : TIMER := (PRE := 4000);   // System Oxidizer Heart Beat Off Timer
   p01r14_oxidizer_heart_beat_ok : BOOL := 1;   // System Oxidizer Heart Beat Ok
   p01r14_oxidizer_heart_beat_on : TIMER := (PRE := 4000, ACC := 152, EN := 1, TT := 1);   // System Oxidizer Heart Beat On Timer
   p01r14_oxidizer_mass_flow : REAL := 4233.082;   // System Oxidizer Oxidizer Mass Flow [SCFM]
   p01r14_timer_fault : TIMER[10] := ([0].PRE := 8000, [1].PRE := 2000, [2].PRE := 1000);   // System Oxidizer Fault Dwell Timer
   p01r14_timer_warning : TIMER[5];
   p02_dint_from_hmi : hmi_dint := (zone_3[6] := 256);
        .HMI[0]   // MOP HMI Iface Dint from HMI Navigation Current Display
        .HMI[1]   // MOP HMI Iface Dint from HMI Navigation PB: Menu Selection
        .HMI[2]   // MOP HMI Iface Dint from HMI Navigation PB: Tab Selection
        .HMI[3]   // MOP HMI Iface Dint from HMI Navigation PB: Page Selection
        .HMI[3].0   // MOP HMI Iface Dint from HMI PB: Next Page
        .HMI[3].1   // MOP HMI Iface Dint from HMI PB: Previous Page
        .HMI[6].30   // MOP HMI Iface Dint from HMI HMI PB: Login
        .HMI[6].31   // MOP HMI Iface Dint from HMI Navigation PB: Clean HMI Screen
        .GLOBAL[0].0   // Dint from HMI Global New Batch Trigger
        .GLOBAL[0].1   // Dint from HMI System PB: Thread Chain Forward
        .GLOBAL[0].2   // Dint from HMI System PB: Thread Slack Take Up
        .GLOBAL[0].3   // Dint from HMI Global Reset Footage Counter
        .GLOBAL[6].0   // MOP HMI Iface Dint from HMI Global PB: Reset Fault
        .GLOBAL[6].1   // MOP HMI Iface Dint from HMI PB: Login
        .GLOBAL[6].2   // MOP HMI Iface Dint from HMI PB: Logout Trigger
        .GLOBAL[6].3   // MOP HMI Iface Dint from HMI Global Reset Maintenance Trigger
        .GLOBAL[6].4   // MOP HMI Iface Dint from HMI Global PB: Line Start
        .GLOBAL[6].5   // MOP HMI Iface Dint from HMI Global PB: Line Stop
        .GLOBAL[6].6   // MOP HMI Iface Dint from HMI Global PB: Line Jog (Not Used)
        .GLOBAL[6].7   // MOP HMI Iface Dint form HMI PB: Stop All Fans
        .GLOBAL[6].10   // MOP HMI Iface Dint to HMI Global PB: Oven Start
        .GLOBAL[6].11   // MOP HMI Iface Dint to HMI Global PB: Oven Stop
        .ZONE_1[4].0   // MOP HMI Iface Dint from HMI Zone 1 Modes PB
        .ZONE_1[4].1   // MOP HMI Iface Dint from HMI Zone 1 Modes PB:
        .ZONE_1[4].2   // MOP HMI Iface Dint from HMI Zone 1 Temperature Control PB:
        .ZONE_1[4].3   // MOP HMI Iface Dint from HMI Zone 1 Temperature Control PB:
        .ZONE_1[4].4   // MOP HMI Iface Dint from HMI Zone 1 Exhaust VFD PB: Start Fan
        .ZONE_1[4].5   // MOP HMI Iface Dint from HMI Zone 1 Exhaust VFD PB: Stop Fan
        .ZONE_1[4].6   // MOP HMI Iface Dint from HMI Zone 1 Exhaust VFD PB: Auto Stop Fan
        .ZONE_1[4].7   // MOP HMI Iface Dint from HMI Zone 1 Recirc VFD PB: Stop Fan
        .ZONE_1[4].8   // MOP HMI Iface Dint from HMI Zone 1 Recirc VFD PB: Start Fan
        .ZONE_1[4].10   // MOP HMI Iface Dint from HMI Zone 1 Recirc VFD PB: Auto Stop Fan
        .ZONE_1[4].12   // MOP HMI Iface Dint from HMI Zone 1
        .ZONE_1[4].13   // MOP HMI Iface Dint from HMI Zone 1
        .ZONE_1[4].14   // MOP HMI Iface Dint from HMI Zone 1
        .ZONE_1[4].16   // MOP HMI Iface Dint from HMI Zone 1 Temperature Control PB: Start Zone Heat Control
        .ZONE_1[4].17   // MOP HMI Iface Dint from HMI Zone 1 Temperature Control PB: Stop Zone Heat Control
        .ZONE_1[4].18   // MOP HMI Iface Dint from HMI Zone 1 Temperature Zone Control PB: Zone Manual Control
        .ZONE_1[4].19   // MOP HMI Iface Dint from HMI Zone 1 Temperature Zone Control PB: Zone Auto Control
        .ZONE_1[4].20   // MOP HMI Iface Dint from HMI Zone 1
        .ZONE_1[4].21   // MOP HMI Iface Dint from HMI Zone 1
        .ZONE_1[4].22   // MOP HMI Iface Dint from HMI Zone 1
        .ZONE_1[4].24   // MOP HMI Iface Dint from HMI Zone 1
        .ZONE_1[4].25   // MOP HMI Iface Dint from HMI Zone 1
        .ZONE_1[4].26   // MOP HMI Iface Dint from HMI Zone 1
        .ZONE_2[4].0   // MOP HMI Iface Dint from HMI Zone 2 Modes PB: Auto Start
        .ZONE_2[4].1   // MOP HMI Iface Dint from HMI Zone 2 Modes PB: Auto Shutdown
        .ZONE_2[4].2   // MOP HMI Iface Dint from HMI Zone 2 Temperature Control PB: Start Chamber Heat Control
        .ZONE_2[4].3   // MOP HMI Iface Dint from HMI Zone 2 Temperature Control PB: Stop Chamber Heat Control
        .ZONE_2[4].4   // MOP HMI Iface Dint from HMI Zone 2 Exhaust VFD PB: Start Fan
        .ZONE_2[4].5   // MOP HMI Iface Dint from HMI Zone 2 Exhaust VFD PB: Stop Fan
        .ZONE_2[4].6   // MOP HMI Iface Dint from HMI Zone 2 Exhaust VFD PB: Auto Stop Fan
        .ZONE_2[4].7   // MOP HMI Iface Dint from HMI Zone 2 Supply VFD PB: Stop Fan
        .ZONE_2[4].8   // MOP HMI Iface Dint from HMI Zone 2 Supply VFD PB: Start Fan
        .ZONE_2[4].10   // MOP HMI Iface Dint from HMI Zone 2 Supply VFD PB: Auto Stop Fan
        .ZONE_2[4].12   // MOP HMI Iface Dint from HMI Zone 2
        .ZONE_2[4].13   // MOP HMI Iface Dint from HMI Zone 2
        .ZONE_2[4].14   // MOP HMI Iface Dint from HMI Zone 2
        .ZONE_2[4].16   // MOP HMI Iface Dint from HMI Zone 2 Temperature Control PB: Start Zone Heat Control
        .ZONE_2[4].17   // MOP HMI Iface Dint from HMI Zone 2 Temperature Control PB: Stop Zone Heat Control
        .ZONE_2[4].18   // MOP HMI Iface Dint from HMI Zone 2 Temperature Control PB: Control Manual
        .ZONE_2[4].19   // MOP HMI Iface Dint from HMI Zone 2 Temperature Control PB: Control Auto
        .ZONE_2[4].20   // MOP HMI Iface Dint from HMI Zone 2
        .ZONE_2[4].21   // MOP HMI Iface Dint from HMI Zone 2
        .ZONE_2[4].22   // MOP HMI Iface Dint from HMI Zone 2
        .ZONE_2[4].24   // MOP HMI Iface Dint from HMI Zone 2
        .ZONE_2[4].25   // MOP HMI Iface Dint from HMI Zone 2
        .ZONE_2[4].26   // MOP HMI Iface Dint from HMI Zone 2
        .ZONE_2[6].0   // MOP HMI Iface Dint from HMI Zone 2 Modes PB: Auto Start
        .ZONE_2[6].1   // MOP HMI Iface Dint from HMI Zone 2 Modes PB: Auto Shutdown
        .ZONE_2[6].2   // MOP HMI Iface Dint from HMI Zone 2 Temperature Control PB: Start Chamber Heat Control
        .ZONE_2[6].3   // MOP HMI Iface Dint from HMI Zone 2 Temperature Control PB: Stop Chamber Heat Control
        .ZONE_2[6].4   // MOP HMI Iface Dint from HMI Zone 2 Exhaust VFD PB: Start Fan
        .ZONE_2[6].5   // MOP HMI Iface Dint from HMI Zone 2 Exhaust VFD PB: Stop Fan
        .ZONE_2[6].6   // MOP HMI Iface Dint from HMI Zone 2 Exhaust VFD PB: Auto Stop Fan
        .ZONE_2[6].8   // MOP HMI Iface Dint from HMI Zone 2 Supply VFD PB: Start Fan
        .ZONE_2[6].9   // MOP HMI Iface Dint from HMI Zone 2 Supply VFD PB: Stop Fan
        .ZONE_2[6].10   // MOP HMI Iface Dint from HMI Zone 2 Supply VFD PB: Auto Stop Fan
        .ZONE_2[6].12   // MOP HMI Iface Dint from HMI Zone 2
        .ZONE_2[6].13   // MOP HMI Iface Dint from HMI Zone 2
        .ZONE_2[6].14   // MOP HMI Iface Dint from HMI Zone 2
        .ZONE_2[6].16   // MOP HMI Iface Dint from HMI Zone 2 Temperature Control PB: Start Zone Heat Control
        .ZONE_2[6].17   // MOP HMI Iface Dint from HMI Zone 2 Temperature Control PB: Stop Zone Heat Control
        .ZONE_2[6].18   // MOP HMI Iface Dint from HMI Zone 2 Temperature Control PB: Toggle Zone Control Auto/Manual
        .ZONE_2[6].20   // MOP HMI Iface Dint from HMI Zone 2
        .ZONE_2[6].21   // MOP HMI Iface Dint from HMI Zone 2
        .ZONE_2[6].22   // MOP HMI Iface Dint from HMI Zone 2
        .ZONE_2[6].24   // MOP HMI Iface Dint from HMI Zone 2
        .ZONE_2[6].25   // MOP HMI Iface Dint from HMI Zone 2
        .ZONE_2[6].26   // MOP HMI Iface Dint from HMI Zone 2
        .ZONE_3[4].0   // MOP HMI Iface Dint from HMI Zone 3 Modes PB: Auto Start
        .ZONE_3[4].1   // MOP HMI Iface Dint from HMI Zone 3 Modes PB: Auto Shutdown
        .ZONE_3[4].2   // MOP HMI Iface Dint from HMI Zone 3 Temperature Control PB: Start Chamber Heat Control
        .ZONE_3[4].3   // MOP HMI Iface Dint from HMI Zone 3 Temperature Control PB: Stop Chamber Heat Control
        .ZONE_3[4].4   // MOP HMI Iface Dint from HMI Zone 3 Exhaust VFD PB: Start Fan
        .ZONE_3[4].5   // MOP HMI Iface Dint from HMI Zone 3 Exhaust VFD PB: Stop Fan
        .ZONE_3[4].6   // MOP HMI Iface Dint from HMI Zone 3 Exhaust VFD PB: Auto Stop Fan
        .ZONE_3[4].7   // MOP HMI Iface Dint from HMI Zone 3 Supply VFD PB: Stop Fan
        .ZONE_3[4].8   // MOP HMI Iface Dint from HMI Zone 3 Supply VFD PB: Start Fan
        .ZONE_3[4].10   // MOP HMI Iface Dint from HMI Zone 3 Supply VFD PB: Auto Stop Fan
        .ZONE_3[4].12   // MOP HMI Iface Dint from HMI Zone 3
        .ZONE_3[4].13   // MOP HMI Iface Dint from HMI Zone 3
        .ZONE_3[4].14   // MOP HMI Iface Dint from HMI Zone 3
        .ZONE_3[4].16   // MOP HMI Iface Dint from HMI Zone 3 Temperature Control PB: Start Zone Heat Control
        .ZONE_3[4].17   // MOP HMI Iface Dint from HMI Zone 3 Temperature Control PB: Stop Zone Heat Control
        .ZONE_3[4].18   // MOP HMI Iface Dint from HMI Zone 3 Temperature Control PB: Toggle Zone Control Manual
        .ZONE_3[4].19   // MOP HMI Iface Dint from HMI Zone 3 Temperature Control PB: Toggle Zone Control Auto
        .ZONE_3[4].20   // MOP HMI Iface Dint from HMI Zone 3
        .ZONE_3[4].21   // MOP HMI Iface Dint from HMI Zone 3
        .ZONE_3[4].22   // MOP HMI Iface Dint from HMI Zone 3
        .ZONE_3[4].24   // MOP HMI Iface Dint from HMI Zone 3
        .ZONE_3[4].25   // MOP HMI Iface Dint from HMI Zone 3
        .ZONE_3[4].26   // MOP HMI Iface Dint from HMI Zone 3
        .ZONE_3[6].0   // MOP HMI Iface Dint from HMI Zone 3 Modes PB: Auto Start
        .ZONE_3[6].1   // MOP HMI Iface Dint from HMI Zone 3 Modes PB: Auto Shutdown
        .ZONE_3[6].2   // MOP HMI Iface Dint from HMI Zone 3 Temperature Control PB: Start Chamber Heat Control
        .ZONE_3[6].3   // MOP HMI Iface Dint from HMI Zone 3 Temperature Control PB: Stop Chamber Heat Control
        .ZONE_3[6].4   // MOP HMI Iface Dint from HMI Zone 3 Exhaust VFD PB: Start Fan
        .ZONE_3[6].5   // MOP HMI Iface Dint from HMI Zone 3 Exhaust VFD PB: Stop Fan
        .ZONE_3[6].6   // MOP HMI Iface Dint from HMI Zone 3 Exhaust VFD PB: Auto Stop Fan
        .ZONE_3[6].8   // MOP HMI Iface Dint from HMI Zone 3 Supply VFD PB: Start Fan
        .ZONE_3[6].9   // MOP HMI Iface Dint from HMI Zone 3 Supply VFD PB: Stop Fan
        .ZONE_3[6].10   // MOP HMI Iface Dint from HMI Zone 3 Supply VFD PB: Auto Stop Fan
        .ZONE_3[6].12   // MOP HMI Iface Dint from HMI Zone 3
        .ZONE_3[6].13   // MOP HMI Iface Dint from HMI Zone 3
        .ZONE_3[6].14   // MOP HMI Iface Dint from HMI Zone 3
        .ZONE_3[6].16   // MOP HMI Iface Dint from HMI Zone 3 Temperature Control PB: Start Zone Heat Control
        .ZONE_3[6].17   // MOP HMI Iface Dint from HMI Zone 3 Temperature Control PB: Stop Zone Heat Control
        .ZONE_3[6].18   // MOP HMI Iface Dint from HMI Zone 3 Temperature Control PB: Toggle Zone Control Auto/Manual
        .ZONE_3[6].20   // MOP HMI Iface Dint from HMI Zone 3
        .ZONE_3[6].21   // MOP HMI Iface Dint from HMI Zone 3
        .ZONE_3[6].22   // MOP HMI Iface Dint from HMI Zone 3
        .ZONE_3[6].24   // MOP HMI Iface Dint from HMI Zone 3
        .ZONE_3[6].25   // MOP HMI Iface Dint from HMI Zone 3
        .ZONE_3[6].26   // MOP HMI Iface Dint from HMI Zone 3
        .LETOFF[0].8   // Main HMI Dint from HMI Accumulator Auto
        .LETOFF[0].9   // Main HMI Dint from HMI PB: Reset Accumulator Sequence
        .LETOFF[0].10   // Main HMI Dint from HMI PB: Accumulator Position Control
        .LETOFF[0].11   // Main HMI Dint from HMI PB: Accumulator Easy Thread
        .UPL[0].0   // Upper Poly Letoff Dint from HMI PB: Letoff A Enable
        .UPL[0].1   // Upper Poly Letoff Dint from HMI PB: Letoff A Disable
        .UPL[0].2   // Upper Poly Letoff Dint from HMI PB: Letoff B Enable
        .UPL[0].3   // Upper Poly Letoff Dint from HMI PB: Letoff B Disable
        .UPL[0].4   // Main HMI Dint from HMI Static Control 1 On
        .UPL[0].5   // Main HMI Dint from HMI Static Control 1 Off
        .LPL[0].0   // Lower Poly Letoff Dint from HMI PB: Letoff A Enable
        .LPL[0].1   // Lower Poly Letoff Dint from HMI PB: Letoff A Disable
        .LPL[0].2   // Lower Poly Letoff Dint from HMI PB: Letoff B Enable
        .LPL[0].3   // Lower Poly Letoff Dint from HMI PB: Letoff B Disable
        .LPL[0].4   // Main HMI Dint from HMI Static Control 1 On
        .LPL[0].5   // Main HMI Dint from HMI Static Control 1 Off
        .WDR[0].4   // Main HMI Dint from HMI Static Control 1 On
        .WDR[0].5   // Main HMI Dint from HMI Static Control 1 Off
        .SPLICE[0].0   // MOP Iface Splice Press Dint from HMI PB: Splice Press Sequencer Reset
        .SPLICE[6].0   // Main HMI Dint from HMI Splice Press PB: Heater On
        .SPLICE[6].1   // Main HMI Dint from HMI Splice Press PB: Heater Off
        .STATIC[0].5   // Main HMI Dint from HMI Static Control 1 Off
        .STATIC[0].9   // Main HMI Dint from HMI Static Control 2 Off
        .STATIC[0].12   // Main HMI Dint from HMI Static Control 3 On
        .MISC[0].0   // Dint from HMI PB: Start Ovens
        .MISC[0].1   // Dint from HMI Stop Ovens
        .EDG[0].0   // Main HMI Dint from HMI PB: Edge Guide On
        .EDG[0].1   // Main HMI Dint from HMI PB: Edge Guide Off
        .EDG[0].2   // Main HMI Dint from HMI PB: Edge Guide Center
        .SLT[1].9   // MOP Iface Dint from HMI PB: Slitter On
        .SLT[1].10   // MOP Iface Dint from HMI PB: Slitter Off
        .IMPREG[0].4   // Main HMI Dint from HMI Static Control 1 On
        .IMPREG[0].5   // Main HMI Dint from HMI Static Control 1 Off
        .IMPREG[0].8   // Main HMI Dint from HMI Static Control 2 On
        .IMPREG[0].9   // Main HMI Dint from HMI Static Control 2 Off
        .IMPREG[0].12   // Main HMI Dint from HMI Static Control 3 On
        .IMPREG[0].13   // Main HMI Dint from HMI Static Control 3 Off
        .IMPREG[0].16   // Impreg Dint from HMI PB: Exhaust Fan Start
        .IMPREG[0].17   // Impreg Dint from HMI PB: Exhaust Fan Stop
        .IMPREG[0].18   // Impreg Dint from HMI PB: Supply Fan Start
        .IMPREG[0].19   // Impreg Dint from HMI PB: Supply Fan Stop
        .IMPREG[0].20   // MOP HMI Iface Dint from HMI PB: Supply Fan Start
        .IMPREG[0].21   // MOP HMI Iface Dint from HMI PB: Supply Fan Stop
        .IMPREG[1].0   // Impreg Dint from HMI PB: Servo Drive Side Jog Forward
        .IMPREG[1].1   // Impreg Dint from HMI PB: Servo Drive Side Jog Reverse
        .IMPREG[1].2   // Impreg Dint from HMI PB: Servo Drive Side Zero
        .IMPREG[1].3   // Impreg Dint from HMI PB: Servo Drive Side Set Offset
        .IMPREG[1].5   // Impreg Dint from HMI PB: Servo Operator Side Jog Forward
        .IMPREG[1].6   // Impreg Dint from HMI PB: Servo Operator Side Jog Reverse
        .IMPREG[1].7   // Impreg Dint from HMI PB: Servo Operator Side Zero
        .IMPREG[1].8   // Impreg Dint from HMI PB: Servo Operator Side Set Offset
        .IMPREG[1].10   // Impreg Dint from HMI PB: Servos to Position Cmd
        .IMPREG[1].12   // Impreg Dint from HMI PB: Servo Drive Side Start
        .IMPREG[1].13   // Impreg Dint from HMI PB: Servo Drive Side Stop
        .IMPREG[1].14   // Impreg Dint from HMI PB: Servo Drive Side Reset
        .IMPREG[1].20   // Impreg Dint from HMI PB: Servo Operator Side Start
        .IMPREG[1].21   // Impreg Dint from HMI PB: Servo Operator Side Stop
        .IMPREG[1].22   // Impreg Dint from HMI PB: Servo Operator Side Reset
        .IMPREG[1].25   // Impgreg Dint from HMI PB: Wet Web Control On
        .ADV_COOLING[4].17   // MOP HMI Iface Dint from HMI Advanced Cooling Temperature Control PB: Zone Control Auto
        .ADV_COOLING[4].18   // MOP HMI Iface Dint from HMI Advanced Cooling Temperature Control PB: Toggle Zone Control Manual
   p02_dint_to_hmi : hmi_dint := (global[0] := 49794, global[1] := 3, global[6] := 260, global[7] := 3, global[8] := 5, global[9] := 1, global[14] := 15533, zone_1[2] := 64, zone_1[4] := 591187, zone_1[5] := 50536423, zone_1[6] := 62708, zone_1[8] := 10, zone_1[9] := 2, zone_1[10] := 2, zone_1[11] := 2, zone_2[4] := 591187, zone_2[5] := 50540519, zone_2[6] := 62708, zone_2[8] := 10, zone_2[9] := 2, zone_2[10] := 2, zone_2[11] := 2, zone_3[4] := 590163, zone_3[5] := 16845924, zone_3[6] := 62708, zone_3[8] := 5, zone_3[9] := 2, zone_3[10] := 2, zone_3[11] := 2, letoff[0] := 37, letoff[1] := 7401712, letoff[4] := 32, letoff[6] := 131072, letoff[7] := 1, ts1[0] := 4, ts1[1] := 4915, ts1[7] := 2, ts2[0] := 983808, ts2[1] := 4915, ts2[6] := 131072, ts2[7] := 2, upl[0] := 5, lpl[0] := 5, wdr[0] := 5, wdr[1] := 5939, wdr[3] := 4785, wdr[4] := 16, wdr[5] := 112, splice[10] := 2, edg[0] := 1, slt[1] := 1136, impreg[0] := 8, impreg[1] := 33879280, impreg[3] := 207668736, impreg[5] := 2, impreg[6] := 2, impreg[7] := 2, impreg[10] := -1, impreg[11] := -1, impreg[12] := -1,
        impreg[13] := -1, adv_cooling[0] := 589840, adv_cooling[1] := 32769, adv_cooling[5] := 16382, retraction[0] := 255);   // MOP HMI Iface Dint to HMI
        .HMI[1]   // MOP HMI Iface Dint from HMI Navigation PI: Menu Selection
        .HMI[2]   // MOP HMI Iface Dint from HMI Navigation PI: Tab Selection
        .HMI[6].31   // MOP HMI Iface Dint from HMI Navigation PI: Clean HMI Screen Done
        .GLOBAL[0].10   // Oxidizer in Heat demand Mode
        .GLOBAL[0].11   // Oxidizer Fault
        .GLOBAL[0].12   // Oven Heat is On
        .GLOBAL[0].13   // Oxidizer at Temperature
        .GLOBAL[0].14   // Ovens are starting
        .GLOBAL[0].15   // Ovens are Stopping
        .GLOBAL[0].16   // LFL High level Warning
        .GLOBAL[0].17   // LFL High level Alarm
        .GLOBAL[0].18   // Static Bar Fault
        .GLOBAL[0].19   // Windup Accumulator at Top LImit
        .GLOBAL[0].20   // Line drive Warning
        .GLOBAL[0].21   // System Faults
        .GLOBAL[0].22   // Impreg Static Bar 1 Need Cleaning
        .GLOBAL[0].23   // Impreg Static Bar 2 Need Cleaning
        .GLOBAL[0].24   // Impreg Static Bar 3 Need Cleaning
        .GLOBAL[0].25   // Upper Poly Static Bar Need Cleaning
        .GLOBAL[0].26   // Lower Poly Static Bar Need Cleaning
        .GLOBAL[0].27   // Laminator Static Bar Need Cleaning
        .GLOBAL[0].28   // Winder Static Bar Need Cleaning
        .LETOFF[0].10   // Main HMI Dint to HMI PI: Accumulator Arm
        .LETOFF[0].11   // Main HMI Dint to HMI PI: Accumulator Disarm
        .WDR[0].0   // Winder A active
        .WDR[0].1   // Winder B active
        .WDR[0].2   // Winder Liner takeup running
        .WDR[0].4   // Static bar Impreg 1 is on
        .WDR[0].5   // Static bar Impreg 1 HVPS is on
        .WDR[0].6   // Static bar Impreg 1 HVPS enabled
        .EDG[0].0   // Edge Control Dint to HMI Edge Guide Auto Mode
   p02_real_from_hmi : hmi_real := (global[1] := 8.0, zone_1[39] := 5.0, zone_1[44] := 50.0, zone_1[47] := 25.0, zone_1[48] := 20.0, zone_1[49] := 1.0, zone_1[51] := 20.0, zone_1[52] := 440.0, zone_1[54] := 20.0, zone_1[55] := 25.0, zone_1[56] := 40.0, zone_1[57] := 110.0, zone_1[58] := -0.25, zone_1[59] := 20.0, zone_1[60] := 20.0, zone_1[68] := 45.0, zone_2[39] := 5.0, zone_2[44] := 50.0, zone_2[47] := 25.0, zone_2[48] := 20.0, zone_2[49] := 0.5, zone_2[51] := 15.0, zone_2[52] := 440.0, zone_2[54] := 20.0, zone_2[55] := 25.0, zone_2[56] := 40.0, zone_2[57] := 122.0, zone_2[58] := -0.25, zone_2[59] := 5.0, zone_2[60] := 15.0, zone_2[68] := 60.0, zone_3[39] := 5.0, zone_3[44] := 10.0, zone_3[45] := 0.1, zone_3[48] := 10.0, zone_3[49] := 1.0, zone_3[52] := 400.0, zone_3[54] := 50.0, zone_3[55] := 25.0, zone_3[56] := 40.0, zone_3[57] := 125.0, zone_3[59] := 5.0, zone_3[60] := 15.0, zone_3[68] := 80.0, letoff[40] := 1.1, letoff[41] := 2.0, letoff[43] := 0.01, ts1[40] := 4.2, ts1[41] := 2.0, ts1[42] := 5.0, ts2[40] := 1.0, ts2[41] := 1.0, wdr[40] := 1.0, wdr[41] := 1.0, wdr[60] := 100.0, wdr[61] := 100.0, splice[44] := 30.0, splice[47] := 30.0, impreg[0] := 0.018, impreg[1] := 0.018,
        impreg[2] := 0.005, impreg[3] := 0.011, impreg[55] := 10.0, impreg[56] := 60.0, impreg[58] := -0.25, adv_cooling[48] := 50.0, adv_cooling[49] := 1.0, adv_cooling[54] := 20.0, adv_cooling[58] := 10.0, adv_cooling[66] := 15.0, adv_cooling[68] := 100.0);   // MOP HMI Iface Real from HMI
        .GLOBAL[1]   // MOP HMI Iface Real from HMI Parameter Master Jog Speed
        .ZONE_1[40]   // MOP HMI Iface Real from HMI Zone 1 Parameter Process Temperature Zero Offset
        .ZONE_1[41]   // MOP HMI Iface Real from HMI Zone 1 Parameter Heater Temperature Zero Offset
        .ZONE_1[42]   // MOP HMI Iface Real from HMI Zone 1 Parameter Spare
        .ZONE_1[43]   // MOP HMI Iface Real from HMI Zone 1 Parameter Spare
        .ZONE_1[44]   // MOP HMI Iface Real from HMI Zone 1 PID1 Kp
        .ZONE_1[45]   // MOP HMI Iface Real from HMI Zone 1 PID1 Ki
        .ZONE_1[46]   // MOP HMI Iface Real from HMI Zone 1 PID1 Kd
        .ZONE_1[47]   // MOP HMI Iface Real from HMI Zone 1 PID1 Bias
        .ZONE_1[48]   // MOP HMI Iface Real from HMI Zone 1 PID2 Kp
        .ZONE_1[49]   // MOP HMI Iface Real from HMI Zone 1 PID2 Ki
        .ZONE_1[50]   // MOP HMI Iface Real from HMI Zone 1 PID2 Kd
        .ZONE_1[51]   // MOP HMI Iface Real from HMI Zone 1 PID2 Bias
        .ZONE_1[52]   // MOP HMI Iface Real from HMI Zone 1 Temperature Control Zone Temperature Process Air High Limit
        .ZONE_1[53]   // MOP HMI Iface Real from HMI Zone 1 Temperature Control Spare
        .ZONE_1[54]   // MOP HMI Iface Real from HMI Zone 1 Temperature Control Zone Temperature Deviation from Setpoin
        .ZONE_1[55]   // MOP HMI Iface Real from HMI Parameter Lower Flash Limit Warning Level
        .ZONE_1[56]   // MOP HMI Iface Real from HMI Parameter Lower Flash Limit Alarm Level
        .ZONE_1[57]   // MOP HMI Iface Real from HMI Parameter Zone Shutdown Temperature
        .ZONE_1[58]   // MOP HMI Iface Real from HMI Parameter Zone Pressure Limit
        .ZONE_1[59]   // MOP HMI Iface Real from HMI Parameter Fast to Soak Deviation
        .ZONE_1[60]   // MOP HMI Iface Real from HMI Parameter Soak to Fast Deviation
        .ZONE_1[61]   // MOP HMI Iface Real from HMI Parameter Spare
        .ZONE_1[62]   // MOP HMI Iface Real from HMI Parameter Spare
        .ZONE_1[63]   // MOP HMI Iface Real from HMI Parameter Spare
        .ZONE_1[64]   // MOP HMI Iface Real from HMI Setpoint Spare
        .ZONE_1[65]   // MOP HMI Iface Real from HMI Setpoint Spare
        .ZONE_1[66]   // MOP HMI Iface Real from HMI Setpoint Spare
        .ZONE_1[67]   // MOP HMI Iface Real from HMI Zone 1 Temperature Control Setpoint
        .ZONE_1[68]   // MOP HMI Iface Real from HMI Zone 1 Temperature Control Manual Heat Control Valve Setpoint
        .ZONE_1[69]   // MOP HMI Iface Real from HMI Setpoint Spare
        .ZONE_1[70]   // MOP HMI Iface Real from HMI Setpoint Spare
        .ZONE_1[71]   // MOP HMI Iface Real from HMI Setpoint Spare
        .ZONE_1[72]   // MOP HMI Iface Real from HMI Zone 1 Temperature Control Process Control Temperature
        .ZONE_1[73]   // MOP HMI Iface Real from HMI Spare
        .ZONE_1[74]   // MOP HMI Iface Real from HMI Spare
        .ZONE_1[75]   // MOP HMI Iface Real from HMI Spare
        .ZONE_1[76]   // MOP HMI Iface Real from HMI Spare
        .ZONE_1[77]   // MOP HMI Iface Real from HMI Spare
        .ZONE_1[78]   // MOP HMI Iface Real from HMI Spare
        .ZONE_1[79]   // MOP HMI Iface Real from HMI Spare
        .ZONE_2[40]   // MOP HMI Iface Real from HMI Zone 2 Parameter Process Temperature Zero Offset
        .ZONE_2[41]   // MOP HMI Iface Real from HMI Zone 2 Parameter Heater Temperature Zero Offset
        .ZONE_2[42]   // MOP HMI Iface Real from HMI Zone 2 Parameter Spare
        .ZONE_2[43]   // MOP HMI Iface Real from HMI Zone 2 Parameter Spare
        .ZONE_2[44]   // MOP HMI Iface Real from HMI Zone 2 PID1 Kp
        .ZONE_2[45]   // MOP HMI Iface Real from HMI Zone 2 PID1 Ki
        .ZONE_2[46]   // MOP HMI Iface Real from HMI Zone 2 PID1 Kd
        .ZONE_2[47]   // MOP HMI Iface Real from HMI Zone 2 PID1 Bias
        .ZONE_2[48]   // MOP HMI Iface Real from HMI Zone 2 PID2 Kp
        .ZONE_2[49]   // MOP HMI Iface Real from HMI Zone 2 PID2 Ki
        .ZONE_2[50]   // MOP HMI Iface Real from HMI Zone 2 PID2 Kd
        .ZONE_2[51]   // MOP HMI Iface Real from HMI Zone 2 PID2 Bias
        .ZONE_2[52]   // MOP HMI Iface Real from HMI Zone 2 Temperature Control Zone Temperature Process Air High Limit
        .ZONE_2[53]   // MOP HMI Iface Real from HMI Zone 2 Temperature Control Spare
        .ZONE_2[54]   // MOP HMI Iface Real from HMI Zone 2 Temperature Control Zone Temperature Deviation from Setpoin
        .ZONE_2[55]   // MOP HMI Iface Real from HMI Parameter Lower Flash Limit Warning Level
        .ZONE_2[56]   // MOP HMI Iface Real from HMI Parameter Lower Flash Limit Alarm Level
        .ZONE_2[57]   // MOP HMI Iface Real from HMI Parameter Zone Shutdown Temperature
        .ZONE_2[58]   // MOP HMI Iface Real from HMI Parameter Zone Pressure Limit
        .ZONE_2[59]   // MOP HMI Iface Real from HMI Parameter Fast to Soak Deviation
        .ZONE_2[60]   // MOP HMI Iface Real from HMI Parameter Soak to Fast Deviation
        .ZONE_2[61]   // MOP HMI Iface Real from HMI Parameter Spare
        .ZONE_2[62]   // MOP HMI Iface Real from HMI Parameter Spare
        .ZONE_2[63]   // MOP HMI Iface Real from HMI Parameter Spare
        .ZONE_2[64]   // MOP HMI Iface Real from HMI Setpoint Spare
        .ZONE_2[65]   // MOP HMI Iface Real from HMI Setpoint Spare
        .ZONE_2[66]   // MOP HMI Iface Real from HMI Setpoint Spare
        .ZONE_2[67]   // MOP HMI Iface Real from HMI Zone 2 Temperature Control Setpoint
        .ZONE_2[68]   // MOP HMI Iface Real from HMI Zone 2 Temperature Control Manual Heat Control Valve Setpoint
        .ZONE_2[69]   // MOP HMI Iface Real from HMI Setpoint Spare
        .ZONE_2[70]   // MOP HMI Iface Real from HMI Setpoint Spare
        .ZONE_2[71]   // MOP HMI Iface Real from HMI Setpoint Spare
        .ZONE_2[72]   // MOP HMI Iface Real from HMI Zone 2 Temperature Control Process Control Temperature
        .ZONE_2[73]   // MOP HMI Iface Real from HMI Spare
        .ZONE_2[74]   // MOP HMI Iface Real from HMI Spare
        .ZONE_2[75]   // MOP HMI Iface Real from HMI Spare
        .ZONE_2[76]   // MOP HMI Iface Real from HMI Spare
        .ZONE_2[77]   // MOP HMI Iface Real from HMI Spare
        .ZONE_2[78]   // MOP HMI Iface Real from HMI Spare
        .ZONE_2[79]   // MOP HMI Iface Real from HMI Spare
        .ZONE_3[40]   // MOP HMI Iface Real from HMI Zone 3 Parameter Process Temperature Zero Offset
        .ZONE_3[41]   // MOP HMI Iface Real from HMI Zone 3 Parameter Heater Temperature Zero Offset
        .ZONE_3[42]   // MOP HMI Iface Real from HMI Zone 3 Parameter Spare
        .ZONE_3[43]   // MOP HMI Iface Real from HMI Zone 3 Parameter Spare
        .ZONE_3[44]   // MOP HMI Iface Real from HMI Zone 3 PID1 Kp
        .ZONE_3[45]   // MOP HMI Iface Real from HMI Zone 3 PID1 Ki
        .ZONE_3[46]   // MOP HMI Iface Real from HMI Zone 3 PID1 Kd
        .ZONE_3[47]   // MOP HMI Iface Real from HMI Zone 3 PID1 Bias
        .ZONE_3[48]   // MOP HMI Iface Real from HMI Zone 3 PID2 Kp
        .ZONE_3[49]   // MOP HMI Iface Real from HMI Zone 3 PID2 Ki
        .ZONE_3[50]   // MOP HMI Iface Real from HMI Zone 3 PID2 Kd
        .ZONE_3[51]   // MOP HMI Iface Real from HMI Zone 3 PID2 Bias
        .ZONE_3[52]   // MOP HMI Iface Real from HMI Zone 3 Temperature Control Zone Temperature Process Air High Limit
        .ZONE_3[53]   // MOP HMI Iface Real from HMI Zone 3 Temperature Control Spare
        .ZONE_3[54]   // MOP HMI Iface Real from HMI Zone 3 Temperature Control Zone Temperature Deviation from Setpoin
        .ZONE_3[55]   // MOP HMI Iface Real from HMI Parameter Lower Flash Limit Warning Level
        .ZONE_3[56]   // MOP HMI Iface Real from HMI Parameter Lower Flash Limit Alarm Level
        .ZONE_3[57]   // MOP HMI Iface Real from HMI Parameter Zone Shutdown Temperature
        .ZONE_3[58]   // MOP HMI Iface Real from HMI Parameter Zone Pressure Limit
        .ZONE_3[59]   // MOP HMI Iface Real from HMI Parameter Fast to Soak Deviation
        .ZONE_3[60]   // MOP HMI Iface Real from HMI Parameter Soak to Fast Deviation
        .ZONE_3[61]   // MOP HMI Iface Real from HMI Parameter Spare
        .ZONE_3[62]   // MOP HMI Iface Real from HMI Parameter Spare
        .ZONE_3[63]   // MOP HMI Iface Real from HMI Parameter Spare
        .ZONE_3[64]   // MOP HMI Iface Real from HMI Setpoint Spare
        .ZONE_3[65]   // MOP HMI Iface Real from HMI Setpoint Spare
        .ZONE_3[66]   // MOP HMI Iface Real from HMI Setpoint Spare
        .ZONE_3[67]   // MOP HMI Iface Real from HMI Zone 3 Temperature Control Setpoint
        .ZONE_3[68]   // MOP HMI Iface Real from HMI Zone 3 Temperature Control Manual Heat Control Valve Setpoint
        .ZONE_3[69]   // MOP HMI Iface Real from HMI Setpoint Spare
        .ZONE_3[70]   // MOP HMI Iface Real from HMI Setpoint Spare
        .ZONE_3[71]   // MOP HMI Iface Real from HMI Setpoint Spare
        .ZONE_3[72]   // MOP HMI Iface Real from HMI Zone 3 Temperature Control Process Control Temperature
        .ZONE_3[73]   // MOP HMI Iface Real from HMI Spare
        .ZONE_3[74]   // MOP HMI Iface Real from HMI Spare
        .ZONE_3[75]   // MOP HMI Iface Real from HMI Spare
        .ZONE_3[76]   // MOP HMI Iface Real from HMI Spare
        .ZONE_3[77]   // MOP HMI Iface Real from HMI Spare
        .ZONE_3[78]   // MOP HMI Iface Real from HMI Spare
        .ZONE_3[79]   // MOP HMI Iface Real from HMI Spare
        .IMPREG[0]   // Main HMI Real to HMI Servo Left Offset
        .IMPREG[1]   // Main HMI Real to HMI Servo Right Offset
        .IMPREG[2]   // Main HMI Real to HMI Servo Jog Velocity
        .IMPREG[3]   // Main HMI Real to HMI Servo Positioning Velocity
        .IMPREG[20]   // MOP HMI Real from HMI Servo Drive Side Velocity Command
        .IMPREG[21]   // MOP HMI Real from HMI Servo Drive Side Jog Velocity Command
        .IMPREG[22]   // MOP HMI Real from HMI Servo Drive Side Position Command
   p02_real_to_hmi : hmi_real := (global[1] := 8.0, global[11] := 210.0, global[12] := 40.0, global[13] := 1583.0, global[14] := 1549.0, global[15] := 250.0, global[16] := 58.0, global[17] := 1557.0, global[18] := 1459.0, global[19] := 4125.5405, zone_1[0] := 260.0, zone_1[1] := 259.7, zone_1[2] := 260.0, zone_1[6] := -0.25, zone_1[8] := 30.891432, zone_1[9] := 4.9, zone_1[10] := 901.0, zone_1[12] := 37.748573, zone_1[13] := 21.9, zone_1[14] := 1101.0, zone_1[24] := 37.48217, zone_1[28] := 900.0, zone_1[30] := 1100.0, zone_1[44] := 50.0, zone_1[47] := 25.0, zone_1[48] := 20.0, zone_1[49] := 1.0, zone_1[51] := 20.0, zone_1[52] := 440.0, zone_1[54] := 20.0, zone_1[55] := 25.0, zone_1[56] := 40.0, zone_1[57] := 110.0, zone_1[58] := -0.25, zone_1[59] := 20.0, zone_1[60] := 20.0, zone_1[67] := 260.0, zone_1[68] := 45.0, zone_1[72] := 260.0, zone_2[0] := 259.80002, zone_2[1] := 260.2, zone_2[2] := 259.80002, zone_2[6] := 0.15795529, zone_2[8] := 30.891432, zone_2[9] := 2.4, zone_2[10] := 901.0, zone_2[14] := 1100.0, zone_2[24] := 34.236786, zone_2[28] := 900.0, zone_2[30] := 1100.0, zone_2[44] := 50.0, zone_2[47] := 25.0, zone_2[48] := 20.0, zone_2[49] := 0.5, zone_2[51] := 15.0, zone_2[52] := 440.0, zone_2[54] := 20.0, zone_2[55] := 25.0, zone_2[56] := 40.0, zone_2[57] := 122.0,
        zone_2[58] := -0.25, zone_2[59] := 5.0, zone_2[60] := 15.0, zone_2[67] := 260.0, zone_2[68] := 60.0, zone_2[72] := 259.80002, zone_3[0] := 61.3, zone_3[1] := 60.600002, zone_3[2] := 61.3, zone_3[8] := 30.891432, zone_3[9] := 0.8, zone_3[10] := 901.0, zone_3[12] := 44.605717, zone_3[13] := 7.4, zone_3[14] := 1301.0, zone_3[24] := 100.0, zone_3[28] := 900.0, zone_3[30] := 1300.0, zone_3[44] := 10.0, zone_3[45] := 0.1, zone_3[48] := 10.0, zone_3[49] := 1.0, zone_3[52] := 400.0, zone_3[54] := 50.0, zone_3[55] := 25.0, zone_3[56] := 40.0, zone_3[57] := 125.0, zone_3[59] := 5.0, zone_3[60] := 15.0, zone_3[67] := 60.0, zone_3[68] := 80.0, zone_3[72] := 61.3, letoff[0] := 153.39998, letoff[1] := 26.143517, letoff[8] := 3.8146973e-06, letoff[14] := -3.8146973e-06, letoff[15] := 65.0, letoff[20] := -3.8146973e-06, letoff[21] := 74.427734, letoff[25] := 10.0, letoff[26] := 32.0, letoff[27] := 32.0, letoff[40] := 1.1, letoff[41] := 2.0, ts1[0] := 58.732376, ts1[40] := 4.2, ts1[41] := 2.0, ts1[42] := 5.0, ts2[0] := 35.082462, ts2[40] := 1.0, ts2[41] := 1.0, upl[0] := 23.032421, upl[1] := 13.867569, lpl[0] := 40.28277, lpl[1] := 16.6, wdr[0] := 72.75, wdr[1] := 31.441757, wdr[3] := 4.6914635, wdr[4] := 3.25, wdr[6] := -0.0024149062,
        wdr[21] := 8736.299, wdr[22] := 70.328125, wdr[40] := 1.0, wdr[41] := 1.0, splice[0] := 66.200005, splice[1] := 55.0, impreg[0] := 0.018, impreg[1] := 0.018, impreg[2] := 0.005, impreg[3] := 0.011, impreg[8] := 3.8146973e-06, impreg[9] := 1199.0, impreg[10] := 0.90000004, impreg[11] := 60.0, impreg[17] := 6553.2, impreg[22] := 0.009000001, impreg[27] := 0.41828796, impreg[28] := -0.00839819, impreg[55] := 10.0, impreg[56] := 60.0, impreg[58] := -0.25, impreg[60] := 0.008100001, impreg[61] := 0.0085, slt[7] := -3.8146973e-06, adv_cooling[0] := 53.9, adv_cooling[1] := 2192.0, adv_cooling[2] := 53.9, adv_cooling[6] := 14.894943, adv_cooling[48] := 50.0, adv_cooling[49] := 1.0, adv_cooling[54] := 20.0, adv_cooling[58] := 10.0, adv_cooling[68] := 100.0, adv_cooling[72] := 53.9, adv_cooling[80] := -1.22e-43, adv_cooling[81] := -1.22e-43, adv_cooling[82] := 2.120817e-38, adv_cooling[83] := 4.90981e-40, adv_cooling[84] := -3.0306319e+13, adv_cooling[85] := 4.54e-43, adv_cooling[86] := 2.2e-44, adv_cooling[87] := 2.5929805e-09, adv_cooling[88] := 6.483587e-10, adv_cooling[89] := 2.8156545e+29, adv_cooling[90] := 1.23412084e+33);   // MOP HMI Iface Real to HMI
        .ZONE_1[16]   // MOP HMI Iface Zone 1 LFL Level
        .ZONE_2[16]   // MOP HMI Iface Zone 2 LFL Level
        .ZONE_3[16]   // MOP HMI Iface Zone 3 LFL Level
        .IMPREG[27]   // MOP HMI Iface Impreg LFL Level
   p02_recipe_from_hmi : recipe := (name := '20210820_rcp.csv', master_line_speed := 10.0, zone_1.recirc_sp := 1100.0, zone_1.exhaust_sp := 900.0, zone_1.temp_sp := 260.0, zone_2.recirc_sp := 1100.0, zone_2.exhaust_sp := 900.0, zone_2.temp_sp := 260.0, zone_3.recirc_sp := 1300.0, zone_3.exhaust_sp := 900.0, zone_3.temp_sp := 60.0, line_speed_sp := 8.0, letoff_tension_sp := 15.0, acc_tension_sp := 50.0, acc_fill_pressure_sp := 10.0, acc_counter_pressure_sp := 10.0, cure_time_sp := 55.0, platen_temp_sp := 450.0, impreg_gap_sp := 0.016, impreg_supply_speed_sp := 1200.0, ts1_tension_sp := 50.0, slitter_speed_sp := 6.0, adv_cooling_temp_sp := 60.0, ts2_tension_sp := 60.0, lower_poly_tension_sp := 2.0, lower_poly_b_tension_sp := 2.0, upper_poly_tension_sp := 2.0, upper_poly_b_tension_sp := 2.0, winder_tension_sp := 70.0, winder_torque_sp := 100.0, tension_deviation_sp := 6.0);   // MOP HMI Iface Recipe From HMI
   p02_recipe_to_hmi : recipe := (name := '20210820_rcp.csv', master_line_speed := 10.0, zone_1.recirc_sp := 1100.0, zone_1.exhaust_sp := 900.0, zone_1.temp_sp := 260.0, zone_2.recirc_sp := 1100.0, zone_2.exhaust_sp := 900.0, zone_2.temp_sp := 260.0, zone_3.recirc_sp := 1300.0, zone_3.exhaust_sp := 900.0, zone_3.temp_sp := 60.0, line_speed_sp := 8.0, letoff_tension_sp := 15.0, acc_tension_sp := 50.0, acc_fill_pressure_sp := 10.0, acc_counter_pressure_sp := 10.0, cure_time_sp := 55.0, platen_temp_sp := 450.0, impreg_gap_sp := 0.016, impreg_supply_speed_sp := 1200.0, ts1_tension_sp := 50.0, slitter_speed_sp := 6.0, adv_cooling_temp_sp := 60.0, ts2_tension_sp := 60.0, lower_poly_tension_sp := 2.0, lower_poly_b_tension_sp := 2.0, upper_poly_tension_sp := 2.0, upper_poly_b_tension_sp := 2.0, winder_tension_sp := 70.0, winder_torque_sp := 100.0, tension_deviation_sp := 6.0);   // MOP HMI Iface To HMI Recipe
   p02r01 : routine := (comment := 7);   // MOP HMI Iface Main
   p02r02 : routine := (comment := -1073741761, oneshot := 1);   // MOP HMI Iface Misc Control
   p02r02_timer_fault : TIMER[4];   // MOP HMI Iface Misc Control Fault Delay
   p02r02_timer_logout : TIMER := (PRE := 900000, ACC := 900000);
   p02r02_timer_warning : TIMER[4];   // MOP HMI Iface Misc Control Warning Delay
   p02r03 : routine := (comment := -1073741793);   // MOP HMI Iface Navigation
   p02r03_timer_fault : TIMER[4];   // MOP HMI Iface Navigation Fault Delay
   p02r03_timer_warning : TIMER[4];   // MOP HMI Iface Navigation Warning Delay
   p02r04 : routine := (comment := -536870835);   // MOP HMI Iface Recipe
   p02r04_timer_fault : TIMER[4];   // MOP HMI Iface Recipe Fault Delay
   p02r04_timer_warning : TIMER[4];   // MOP HMI Iface Recipe Warning Delay
   p02r05 : routine := (comment := -1073741729);   // MOP HMI Iface Dint to HMI
   p02r05_timer_fault : TIMER[4];   // MOP HMI Iface Dint to HMI Fault Delay
   p02r05_timer_warning : TIMER[4];   // MOP HMI Iface Dint to HMI Warning Delay
   p02r06 : routine := (comment := -1073737569);   // MOP HMI Iface Real to HMI
   p02r06_timer_fault : TIMER[4];   // MOP HMI Iface Real to HMI Fault Delay
   p02r06_timer_warning : TIMER[4];   // MOP HMI Iface Real to HMI Warning Delay
   p02r07 : routine := (comment := -1073737721);   // MOP HMI Iface Alarms
   p02r07_timer_fault : TIMER[4];   // MOP HMI Iface Alarms Fault Delay
   p02r07_timer_warning : TIMER[4];   // MOP HMI Iface Alarms Warning Delay
   p02r08 : routine := (comment := -1073741817);   // MOP HMI Iface Warnings
   p02r08_timer_fault : TIMER[4];   // MOP HMI Iface Warnings Fault Delay
   p02r08_timer_warning : TIMER[4];   // MOP HMI Iface Warnings Warning Delay
   p02r09 : routine := (comment := -1073741761);   // MOP HMI Iface Maintenance
   p02r09_timer_fault : TIMER[4];   // MOP HMI Iface Maintenance Fault Delay
   p02r09_timer_warning : TIMER[4];   // MOP HMI Iface Maintenance Warning Delay
   p02r10 : routine := (comment := -1073741761);   // MOP HMI Iface
   p02r10_timer_fault : TIMER[4];   // MOP HMI Iface Fault Delay
   p02r10_timer_warning : TIMER[4];   // MOP HMI Iface Warning Delay
   p02r11 : routine := (comment := -1073741761);   // MOP HMI Iface
   p02r11_timer_fault : TIMER[4];   // MOP HMI Iface Fault Delay
   p02r11_timer_warning : TIMER[4];   // MOP HMI Iface Warning Delay
   p02r12 : routine := (comment := -1073741761);   // MOP HMI Iface
   p02r12_timer_fault : TIMER[4];   // MOP HMI Iface Fault Delay
   p02r12_timer_warning : TIMER[4];   // MOP HMI Iface Warning Delay
   p02r13 : routine := (comment := -1073741761);   // MOP HMI Iface
   p02r13_timer_fault : TIMER[4];   // MOP HMI Iface Fault Delay
   p02r13_timer_warning : TIMER[4];   // MOP HMI Iface Warning Delay
   p02r14 : routine := (comment := -1073741761);   // MOP HMI Iface
   p02r14_timer_fault : TIMER[4];   // MOP HMI Iface Fault Delay
   p02r14_timer_warning : TIMER[4];   // MOP HMI Iface Warning Delay
   p02r15 : routine := (comment := -1073741761);   // MOP HMI Iface
   p02r15_timer_fault : TIMER[4];   // MOP HMI Iface Fault Delay
   p02r15_timer_warning : TIMER[4];   // MOP HMI Iface Warning Delay
   p11_ai_exh_amps : REAL := 4.9;   // Zone 1 Analog Input Exhaust Fan Amps
   p11_ai_exh_hz : REAL := 30.891432;   // Zone 1 Analog Input Exhaust Fan HZ
   p11_ai_exh_hz_max : REAL := 60.0;   // Zone 1 Analog Inputs Exhaust VFD max Hz
   p11_ai_exh_pct : REAL;   // Zone 1 Analog Input Exhaust Fan PCT
   p11_ai_exh_rpm : REAL := 901.0;   // Zone 1 Analog Input Exhaust Fan RPM
   p11_ai_lfl : REAL;   // Zone 1 Analog Input Lower Flash Limit
   p11_ai_prs : REAL := -0.25;   // Zone 1 Analog Input Pressure
   p11_ai_recirc_amps : REAL := 21.9;   // Zone 1 Analog Input Recirc Fan Amps
   p11_ai_recirc_hz : REAL := 37.748573;   // Zone 1 Analog Input Supply Fan HZ
   p11_ai_recirc_hz_max : REAL := 60.0;   // Zone 1 Analog Inputs Recric Fan Max Hz
   p11_ai_recirc_pct : REAL;   // Zone 1 Analog Input Recirc Fan PCT
   p11_ai_recirc_rpm : REAL := 1101.0;   // Zone 1 Analog Input Recirc Fan RPM
   p11_ai_tc01 : REAL := 260.0;   // Zone 1 Analog Input Control Thermocouple 1
   p11_ai_tc02 : REAL := 259.7;   // Zone 1 Analog Input Control Thermocouple 2
   p11_ao_cv : REAL := 37.48217;   // Zone 1 Analog Output Control Valve
   p11_ao_exhaust_selected_speed : REAL := 900.0;   // Zone 1 Analog Output Exhaust Fan VFD Selected Speed
   p11_ao_recirc_selected_speed : REAL := 1100.0;   // Zone 1 Analog Output Recirc Fan VFD Selected Speed
   p11_di_burner_auto : BOOL := 1;   // Zone 1 Digital Input Burner Auto
   p11_di_burner_safeties_ok : BOOL := 1;   // Zone 1 Digital Input Burner Safeties Ok
   p11_di_door_open : BOOL;   // Zone 1 Digital Input Access Door Open
   p11_di_exh : acs800_di_normal := (running_fwd := 1, ready := 1, ctrl_from_net := 1, ref_from_net := 1, at_reference := 1);   // Zone 1 Digital Inputs Exhaust Fan
        .FAULTED   // Zone 1 Digital Inputs Exhaust Fan
   p11_di_exh_fan_mtr_ts : BOOL := 1;   // Zone 1 Digital Input Exhaust Fan Motor Thermostat OK
   p11_di_exh_flow_ok : BOOL := 1;   // Zone 1 Digital Input Exhaust Flow OK
   p11_di_flame_failure : BOOL;   // Zone 1 Digital Input Flame Failure
   p11_di_flame_on : BOOL := 1;   // Zone 1 Digital Input Burner is On
   p11_di_fresh_air_clean : BOOL;   // Zone 1 Digital Input Fresh Air Filter Dirty
   p11_di_high_limit_temp_ok : BOOL := 1;   // Zone 1 Digital Input High Limit Temperature OK
   p11_di_recirc : acs800_di_normal := (running_fwd := 1, ready := 1, ctrl_from_net := 1, ref_from_net := 1, at_reference := 1);   // Zone 1 Digital Inputs Recirc Fan
   p11_di_recirc_fan_mtr_ts : BOOL := 1;   // Zone 1 Digital Input Recirc Fan Motor Thermostat OK
   p11_di_recirc_flow_ok : BOOL := 1;   // Zone 1 Digital Input Recirc Flow OK
   p11_di_sp0 : BOOL;   // Zone 1 Digital Input Combustion Blower Pressure OK
   p11_di_sp00 : BOOL;   // Zone 1 Digital Input Recirculation Air Filter Dirty
   p11_di_sp1 : BOOL;
   p11_di_sp2 : BOOL;
   p11_di_sp3 : BOOL;
   p11_di_tc01_bo : BOOL;   // Zone 1 Digital Input Control Thermocouple 1 Failure
   p11_di_tc02_bo : BOOL;   // Zone 1 Digital Input Control Thermocouple 2 Failure
   p11_di_zone_air_clean : BOOL := 1;   // Zone 1 Digital Input Combustion Air Filter Dirty
   p11_dint_to_hmi : DINT[16] := ([2] := 64, [4] := 591187, [5] := 50536423, [6] := 62708, [8] := 10, [9] := 2, [10] := 2, [11] := 2);   // Zone 1 Temperature Control VFDs On
        [0]   // Zone 1 Dint to HMI Alarms
        [0].0   // Zone 1 Dint to HMI Alarms A00: Process Control Software High Limit
        [0].1   // Zone 1 Dint to HMI Alarms A01: Process Control Hardware High Limit
        [0].2   // Zone 1 Dint to HMI Alarms A02: Process Control Thermocouple Failure
        [0].3   // Zone 1 Dint to HMI Alarms A03: Process Control Temperature Spare
        [0].4   // Zone 1 Dint to HMI Alarms A04: Lower Flash Limit High High Limit Exceeded
        [0].5   // Zone 1 Dint to HMI Alarms A05: Flame Failure
        [0].6   // Zone 1 Dint to HMI Alarms A06: Burner Safeties Failure
        [0].7   // Zone 1 Dint to HMI Alarms A07: Recirculation Fan Speed Fault
        [0].8   // Zone 1 Dint to HMI Alarms A08: Exhaust Fan Speed Fault
        [0].9   // Zone 1 Dint to HMI Alarms A09: Access Door Open
        [0].10   // Zone 1 Dint to HMI Alarms A10:
        [0].11   // Zone 1 Dint to HMI Alarms A11:
        [0].12   // Zone 1 Dint to HMI Alarms A12:
        [0].13   // Zone 1 Dint to HMI Alarms A13:
        [0].14   // Zone 1 Dint to HMI Alarms A14:
        [0].15   // Zone 1 Dint to HMI Alarms A15:
        [0].16   // Zone 1 Dint to HMI Alarms A16: Exhaust Fan Drive Fault
        [0].17   // Zone 1 Dint to HMI Alarms A17: Exhaust Fan Motor Thermistor Not OK
        [0].18   // Zone 1 Dint to HMI Alarms A18: Exhaust Fan VFD Not Ready
        [0].19   // Zone 1 Dint to HMI Alarms A19:
        [0].20   // Zone 1 Dint to HMI Alarms A20: Recirculation Fan Drive Fault
        [0].21   // Zone 1 Dint to HMI Alarms A21: Recirculation Fan Motor Thermistor Not OK
        [0].22   // Zone 1 Dint to HMI Alarms A22: Recirculation Fan VFD Not Ready
        [0].23   // Zone 1 Dint to HMI Alarms A23:
        [0].24   // Zone 1 Dint to HMI Alarms A24:
        [0].25   // Zone 1 Dint to HMI Alarms A25:
        [0].26   // Zone 1 Dint to HMI Alarms A26:
        [0].27   // Zone 1 Dint to HMI Alarms A27:
        [0].28   // Zone 1 Dint to HMI Alarms A28:
        [0].29   // Zone 1 Dint to HMI Alarms A29:
        [0].30   // Zone 1 Dint to HMI Alarms A30:
        [0].31   // Zone 1 Dint to HMI Alarms A31:
        [1]   // Zone 1 Dint to HMI Alarms
        [1].0   // Zone 1 Dint to HMI Alarms
        [1].1   // Zone 1 Dint to HMI Alarms
        [1].2   // Zone 1 Dint to HMI Alarms
        [1].3   // Zone 1 Dint to HMI Alarms
        [1].4   // Zone 1 Dint to HMI Alarms
        [1].5   // Zone 1 Dint to HMI Alarms
        [1].6   // Zone 1 Dint to HMI Alarms
        [1].7   // Zone 1 Dint to HMI Alarms
        [1].8   // Zone 1 Dint to HMI Alarms
        [1].9   // Zone 1 Dint to HMI Alarms
        [1].10   // Zone 1 Dint to HMI Alarms
        [1].11   // Zone 1 Dint to HMI Alarms
        [1].12   // Zone 1 Dint to HMI Alarms
        [1].13   // Zone 1 Dint to HMI Alarms
        [1].14   // Zone 1 Dint to HMI Alarms
        [1].15   // Zone 1 Dint to HMI Alarms
        [1].16   // Zone 1 Dint to HMI Alarms
        [1].17   // Zone 1 Dint to HMI Alarms
        [1].18   // Zone 1 Dint to HMI Alarms
        [1].19   // Zone 1 Dint to HMI Alarms
        [1].20   // Zone 1 Dint to HMI Alarms
        [1].21   // Zone 1 Dint to HMI Alarms
        [1].22   // Zone 1 Dint to HMI Alarms
        [1].23   // Zone 1 Dint to HMI Alarms
        [1].24   // Zone 1 Dint to HMI Alarms
        [1].25   // Zone 1 Dint to HMI Alarms
        [1].26   // Zone 1 Dint to HMI Alarms
        [1].27   // Zone 1 Dint to HMI Alarms
        [1].28   // Zone 1 Dint to HMI Alarms
        [1].29   // Zone 1 Dint to HMI Alarms
        [1].30   // Zone 1 Dint to HMI Alarms
        [1].31   // Zone 1 Dint to HMI Alarms
        [2]   // Zone 1 Dint to HMI Warnings
        [2].0   // Zone 1 Dint to HMI Warnings W00: Control Temperature Deviation
        [2].1   // Zone 1 Dint to HMI Warnings W01: Process Control Thermocouple 1 Failure
        [2].2   // Zone 1 Dint to HMI Warnings W02: Process Control Thermocouple 2 Failure
        [2].3   // Zone 1 Dint to HMI Warnings W03: Control Valve in Manual
        [2].4   // Zone 1 Dint to HMI Warnings W04: LFL High Limit
        [2].5   // Zone 1 Dint to HMI Warnings W05: Zone Off
        [2].6   // Zone 1 Dint to HMI Warnings W06: Fresh Air Filter Dirty
        [2].7   // Zone 1 Dint to HMI Warnings W07: Combustion Air Filter Dirty
        [2].8   // Zone 1 Dint to HMI Warnings W08: Recirculation Air Filter Dirty
        [2].9   // Zone 1 Dint to HMI Warnings W09:
        [2].10   // Zone 1 Dint to HMI Warnings W10:
        [2].11   // Zone 1 Dint to HMI Warnings W11:
        [2].12   // Zone 1 Dint to HMI Warnings W12:
        [2].13   // Zone 1 Dint to HMI Warnings W13:
        [2].14   // Zone 1 Dint to HMI Warnings W14:
        [2].15   // Zone 1 Dint to HMI Warnings W15: Low Pressure
        [2].16   // Zone 1 Dint to HMI Warnings W16: Exhaust Fan Stopped While Zone is Too Hot
        [2].17   // Zone 1 Dint to HMI Warnings W17: Fan Flow Failure
        [2].18   // Zone 1 Dint to HMI Warnings W18: Exhaust VFD Warning
        [2].19   // Zone 1 Dint to HMI Warnings W19:
        [2].20   // Zone 1 Dint to HMI Warnings W20: Recirculation Fan Stopped While Zone is Too Hot
        [2].21   // Zone 1 Dint to HMI Warnings W21: Recirculation Fan Flow Failure
        [2].22   // Zone 1 Dint to HMI Warnings W22:
        [2].23   // Zone 1 Dint to HMI Warnings W23:
        [2].24   // Zone 1 Dint to HMI Warnings W24:
        [2].25   // Zone 1 Dint to HMI Warnings W25:
        [2].26   // Zone 1 Dint to HMI Warnings W26:
        [2].27   // Zone 1 Dint to HMI Warnings W27:
        [2].28   // Zone 1 Dint to HMI Warnings W28:
        [2].29   // Zone 1 Dint to HMI Warnings W29:
        [2].30   // Zone 1 Dint to HMI Warnings W30:
        [2].31   // Zone 1 Dint to HMI Warnings W31:
        [3]   // Zone 1 Dint to HMI Warnings
        [3].0   // Zone 1 Dint to HMI Alarms
        [3].1   // Zone 1 Dint to HMI Alarms
        [3].2   // Zone 1 Dint to HMI Alarms
        [3].3   // Zone 1 Dint to HMI Alarms
        [3].4   // Zone 1 Dint to HMI Alarms
        [3].5   // Zone 1 Dint to HMI Alarms
        [3].6   // Zone 1 Dint to HMI Alarms
        [3].7   // Zone 1 Dint to HMI Alarms
        [3].8   // Zone 1 Dint to HMI Alarms
        [3].9   // Zone 1 Dint to HMI Alarms
        [3].10   // Zone 1 Dint to HMI Alarms
        [3].11   // Zone 1 Dint to HMI Alarms
        [3].12   // Zone 1 Dint to HMI Alarms
        [3].13   // Zone 1 Dint to HMI Alarms
        [3].14   // Zone 1 Dint to HMI Alarms
        [3].15   // Zone 1 Dint to HMI Alarms
        [3].16   // Zone 1 Dint to HMI Alarms
        [3].17   // Zone 1 Dint to HMI Alarms
        [3].18   // Zone 1 Dint to HMI Alarms
        [3].19   // Zone 1 Dint to HMI Alarms
        [3].20   // Zone 1 Dint to HMI Alarms
        [3].21   // Zone 1 Dint to HMI Alarms
        [3].22   // Zone 1 Dint to HMI Alarms
        [3].23   // Zone 1 Dint to HMI Alarms
        [3].24   // Zone 1 Dint to HMI Alarms
        [3].25   // Zone 1 Dint to HMI Alarms
        [3].26   // Zone 1 Dint to HMI Alarms
        [3].27   // Zone 1 Dint to HMI Alarms
        [3].28   // Zone 1 Dint to HMI Alarms
        [3].29   // Zone 1 Dint to HMI Alarms
        [3].30   // Zone 1 Dint to HMI Alarms
        [3].31   // Zone 1 Dint to HMI Alarms
        [4]   // Zone 1 Dint to HMI Process Indicators
        [4].0   // Zone 1 Dint to HMI PI: Zone Fault
        [4].1   // Zone 1 Dint to HMI PI: VFDs Ready/OK
        [4].2   // Zone 1 Dint to HMI PI:
        [4].3   // Zone 1 Dint to HMI PI:
        [4].4   // Zone 1 Dint to HMI Exhaust VFD PI: Request Auto Run
        [4].5   // Zone 1 Dint to HMI Exhaust VFD PI: VFD Stopped
        [4].6   // Zone 1 Dint to HMI Exhaust VFD PI: Request Auto Stop
        [4].7   // Zone 1 Dint to HMI Exhaust VFD PI:
        [4].8   // Zone 1 Dint to HMI Recirc VFD PI: Request Auto Run
        [4].9   // Zone 1 Dint to HMI Recirc VFD PI: VFD Stopped
        [4].10   // Zone 1 Dint to HMI Recirc VFD PI: Request Auto Stop
        [4].11   // Zone 1 Dint to HMI Supply VFD PI:
        [4].12   // Zone 1 Dint to HMI PI:
        [4].13   // Zone 1 Dint to HMI PI:
        [4].14   // Zone 1 Dint to HMI PI:
        [4].15   // Zone 1 Dint to HMI PI:
        [4].16   // Zone 1 Dint to HMI Temperature Control PI: Request Heat
        [4].17   // Zone 1 Dint to HMI Temperature Control PI: Off
        [4].18   // Zone 1 Dint to HMI Temperature Control PI: Request Manual Control
        [4].19   // Zone 1 Dint to HMI Temperature Control PI: Request Auto Control
        [4].20   // Zone 1 Dint to HMI PI:
        [4].21   // Zone 1 Dint to HMI PI:
        [4].22   // Zone 1 Dint to HMI PI:
        [4].23   // Zone 1 Dint to HMI PI:
        [4].24   // Zone 1 Dint to HMI PI:
        [4].25   // Zone 1 Dint to HMI PI:
        [4].26   // Zone 1 Dint to HMI PI:
        [4].27   // Zone 1 Dint to HMI PI:
        [4].28   // Zone 1 Dint to HMI PI:
        [4].29   // Zone 1 Dint to HMI PI:
        [4].30   // Zone 1 Dint to HMI PI:
        [4].31   // Zone 1 Dint to HMI PI:
        [5]   // Zone 1 Dint to HMI Process Indicators
        [5].0   // Zone 1 Dint to HMI PI: Digital Input Burner Auto
        [5].1   // Zone 1 Dint to HMI PI: Digital Input Burner Safeties Ok
        [5].2   // Zone 1 Dint to HMI PI: Digital Input Combustion Air Filter Clean
        [5].3   // Zone 1 Dint to HMI PI: Digital Input Combustion Blower Pressure OK
        [5].4   // Zone 1 Dint to HMI PI: Digital Input Access Door Open
        [5].5   // Zone 1 Dint to HMI PI: Digital Input Exhaust Fan Motor Thermostat OK
        [5].6   // Zone 1 Dint to HMI PI: Digital Input Exhaust Flow OK
        [5].7   // Zone 1 Dint to HMI PI: Digital Input Flame Failure
        [5].8   // Zone 1 Dint to HMI PI: Digital Input Burner is On
        [5].9   // Zone 1 Dint to HMI PI: Digital Input High Limit Temperature OK
        [5].10   // Zone 1 Dint to HMI PI: Digital Input Recirc Fan Motor Thermostat OK
        [5].11   // Zone 1 Dint to HMI PI: Digital Input Recirc Flow OK
        [5].12   // Zone 1 Dint to HMI PI: Digital Input Recirculation Air Filter Clean
        [5].13   // Zone 1 Dint to HMI PI: Digital Input Fresh Air Filter Clean
        [5].14   // Zone 1 Dint to HMI PI: Digital Input Control Thermocouple 1 Failure
        [5].15   // Zone 1 Dint to HMI PI: Digital Input Control Thermocouple 2 Failure
        [5].16   // Zone 1 Dint to HMI PI: Digital Input Exhaust Fan Running Fwd
        [5].24   // Zone 1 Dint to HMI PI: Digital Input Recirculation Fan Running Fwd
        [6]   // Zone 1 Dint to HMI
        [6].0   // Zone 1 Dint to HMI Exhaut VFD Faulted
        [6].1   // Zone 1 Dint to HMI Exhaut VFD Warning
        [6].2   // Zone 1 Dint to HMI Exhaut VFD Running Forward
        [6].3   // Zone 1 Dint to HMI Exhaut VFD Running Reverse
        [6].4   // Zone 1 Dint to HMI Exhaut VFD Ready
        [6].5   // Zone 1 Dint to HMI Exhaut VFD Control from Net
        [6].6   // Zone 1 Dint to HMI Exhaut VFD Reference from Net
        [6].7   // Zone 1 Dint to HMI Exhaut VFD at Reference
        [6].8   // Zone 1 Dint to HMI Recirc VFD Faulted
        [6].9   // Zone 1 Dint to HMI Recirc VFD Warning
        [6].10   // Zone 1 Dint to HMI Recirc VFD Running Forward
        [6].11   // Zone 1 Dint to HMI Recirc VFD Running Reverse
        [6].12   // Zone 1 Dint to HMI Recirc VFD Ready
        [6].13   // Zone 1 Dint to HMI Recirc VFD Control from Net
        [6].14   // Zone 1 Dint to HMI Recirc VFD Reference from Net
        [6].15   // Zone 1 Dint to HMI Recirc VFD At Reference
        [6].16   // Zone 1 Dint to HMI Temperature Control PI: Request Heat
        [6].17   // Zone 1 Dint to HMI Temperature Control PI: Off
        [6].18   // Zone 1 Dint to HMI Temperature Control PI: Request Manual Control
        [6].19   // Zone 1 Dint to HMI Temperature Control PI:
        [6].20   // Zone 1 Dint to HMI PI:
        [6].21   // Zone 1 Dint to HMI PI:
        [6].22   // Zone 1 Dint to HMI PI:
        [6].23   // Zone 1 Dint to HMI PI:
        [6].24   // Zone 1 Dint to HMI PI:
        [6].25   // Zone 1 Dint to HMI PI:
        [6].26   // Zone 1 Dint to HMI PI:
        [6].27   // Zone 1 Dint to HMI PI:
        [6].28   // Zone 1 Dint to HMI PI:
        [6].29   // Zone 1 Dint to HMI PI:
